LIN {X 0,Y 211.438,Z 626.963,A -85,B 0,C 180,E1 -20790,E2 -20790} C_VEL
LIN {X 0,Y 211.437,Z 626.323,A -85,B 0,C 180,E1 -20793.812,E2 -20793.812} C_VEL
LIN {X 0,Y 211.828,Z 624.336,A -85,B 0,C 180,E1 -20797.626,E2 -20797.626} C_VEL
LIN {X 0,Y 212.751,Z 620.963,A -85,B 0,C 180,E1 -20801.432,E2 -20801.432} C_VEL
LIN {X 0,Y 214.27,Z 616.102,A -85,B 0,C 180,E1 -20805.212,E2 -20805.212} C_VEL
LIN {X 0,Y 216.148,Z 611.384,A -85,B 0,C 180,E1 -20807.992,E2 -20807.992} C_VEL
LIN {X 0,Y 218.416,Z 604.89,A -85,B 0,C 180,E1 -20811.07,E2 -20811.07} C_VEL
LIN {X 0,Y 221.135,Z 597.399,A -85,B 0,C 180,E1 -20813.905,E2 -20813.905} C_VEL
LIN {X 0,Y 224.235,Z 588.787,A -85,B 0,C 180,E1 -20816.527,E2 -20816.527} C_VEL
LIN {X 0,Y 227.75,Z 578.349,A -85,B 0,C 180,E1 -20819.079,E2 -20819.079} C_VEL
LIN {X 0,Y 231.118,Z 567.814,A -85,B 0,C 180,E1 -20821.128,E2 -20821.128} C_VEL
LIN {X 0,Y 234.172,Z 556.322,A -85,B 0,C 180,E1 -20822.954,E2 -20822.954} C_VEL
LIN {X 0,Y 234.795,Z 553.459,A -85,B 0,C 180,E1 -20823.368,E2 -20823.368} C_VEL
LIN {X 0,Y 234.361,Z 541.271,A -85,B 0,C 180,E1 -20825.351,E2 -20825.351} C_VEL
LIN {X 0,Y 232.923,Z 528.444,A -85,B 0,C 180,E1 -20827.232,E2 -20827.232} C_VEL
LIN {X 0,Y 230.563,Z 516.355,A -85,B 0,C 180,E1 -20828.886,E2 -20828.886} C_VEL
LIN {X 0,Y 227.516,Z 504.968,A -85,B 0,C 180,E1 -20830.356,E2 -20830.356} C_VEL
LIN {X 0,Y 222.858,Z 491.263,A -85,B 0,C 180,E1 -20832.099,E2 -20832.099} C_VEL
LIN {X 0,Y 223.254,Z 487.862,A -85,B 0,C 180,E1 -20833.833,E2 -20833.833} C_VEL
LIN {X 0,Y 222.449,Z 481.719,A -85,B 0,C 180,E1 -20837.469,E2 -20837.469} C_VEL
LIN {X 0,Y 221.31,Z 475.041,A -85,B 0,C 180,E1 -20841.74,E2 -20841.74} C_VEL
LIN {X 0,Y 220.41,Z 470.31,A -85,B 0,C 180,E1 -20844.974,E2 -20844.974} C_VEL
LIN {X 0,Y 219.512,Z 466.3,A -85,B 0,C 180,E1 -20847.926,E2 -20847.926} C_VEL
LIN {X 0,Y 222.724,Z 476.254,A -85,B 0,C 180,E1 -20849.677,E2 -20849.677} C_VEL
LIN {X 0,Y 225.072,Z 485.139,A -85,B 0,C 180,E1 -20851.347,E2 -20851.347} C_VEL
LIN {X 0,Y 222.609,Z 498.639,A -85,B 0,C 180,E1 -20853.769,E2 -20853.769} C_VEL
LIN {X 0,Y 220.199,Z 511.207,A -85,B 0,C 180,E1 -20856.487,E2 -20856.487} C_VEL
LIN {X 0,Y 217.759,Z 523.017,A -85,B 0,C 180,E1 -20859.555,E2 -20859.555} C_VEL
LIN {X 0,Y 216.268,Z 532.38,A -85,B 0,C 180,E1 -20862.506,E2 -20862.506} C_VEL
LIN {X 0,Y 214.739,Z 541.158,A -85,B 0,C 180,E1 -20865.791,E2 -20865.791} C_VEL
LIN {X 0,Y 213.615,Z 549.495,A -85,B 0,C 180,E1 -20869.575,E2 -20869.575} C_VEL
LIN {X 0,Y 213.008,Z 556.211,A -85,B 0,C 180,E1 -20873.369,E2 -20873.369} C_VEL
LIN {X 0,Y 212.724,Z 561.483,A -85,B 0,C 180,E1 -20877.159,E2 -20877.159} C_VEL
LIN {X 0,Y 212.687,Z 564.579,A -85,B 0,C 180,E1 -20880,E2 -20880} C_VEL
LIN {X 0,Y 213.289,Z 567.702,A -85,B 0,C 180,E1 -20883.778,E2 -20883.778} C_VEL
LIN {X 0,Y 214.604,Z 569.684,A -85,B 0,C 180,E1 -20887.527,E2 -20887.527} C_VEL
LIN {X 0,Y 216.505,Z 570.581,A -85,B 0,C 180,E1 -20891.231,E2 -20891.231} C_VEL
LIN {X 0,Y 218.953,Z 570.405,A -85,B 0,C 180,E1 -20894.879,E2 -20894.879} C_VEL
LIN {X 0,Y 222.069,Z 569.211,A -85,B 0,C 180,E1 -20898.45,E2 -20898.45} C_VEL
LIN {X 0,Y 226.094,Z 566.97,A -85,B 0,C 180,E1 -20901.901,E2 -20901.901} C_VEL
LIN {X 0,Y 230.851,Z 563.736,A -85,B 0,C 180,E1 -20905.227,E2 -20905.227} C_VEL
LIN {X 0,Y 236.622,Z 559.339,A -85,B 0,C 180,E1 -20908.374,E2 -20908.374} C_VEL
LIN {X 0,Y 244.707,Z 552.327,A -85,B 0,C 180,E1 -20912.095,E2 -20912.095} C_VEL
LIN {X 0,Y 251.951,Z 545.424,A -85,B 0,C 180,E1 -20914.878,E2 -20914.878} C_VEL
LIN {X 0,Y 261.05,Z 536.046,A -85,B 0,C 180,E1 -20917.769,E2 -20917.769} C_VEL
LIN {X 0,Y 264.355,Z 532.395,A -85,B 0,C 180,E1 -20918.706,E2 -20918.706} C_VEL
LIN {X 0,Y 264.555,Z 531.824,A -85,B 0,C 180,E1 -20919.611,E2 -20919.611} C_VEL
LIN {X 0,Y 263.168,Z 532.972,A -85,B 0,C 180,E1 -20921.427,E2 -20921.427} C_VEL
LIN {X 0,Y 262.284,Z 533.945,A -85,B 0,C 180,E1 -20922.232,E2 -20922.232} C_VEL
LIN {X 0,Y 260.132,Z 536.442,A -85,B 0,C 180,E1 -20923.31,E2 -20923.31} C_VEL
LIN {X 0,Y 257.399,Z 539.583,A -85,B 0,C 180,E1 -20924.267,E2 -20924.267} C_VEL
LIN {X 0,Y 251.606,Z 546.399,A -85,B 0,C 180,E1 -20926.185,E2 -20926.185} C_VEL
LIN {X 0,Y 250.054,Z 548.43,A -85,B 0,C 180,E1 -20926.914,E2 -20926.914} C_VEL
LIN {X 0,Y 246.157,Z 553.947,A -85,B 0,C 180,E1 -20928.954,E2 -20928.954} C_VEL
LIN {X 0,Y 241.773,Z 559.648,A -85,B 0,C 180,E1 -20930.784,E2 -20930.784} C_VEL
LIN {X 0,Y 234.168,Z 569.412,A -85,B 0,C 180,E1 -20934.129,E2 -20934.129} C_VEL
LIN {X 0,Y 230.572,Z 573.702,A -85,B 0,C 180,E1 -20935.675,E2 -20935.675} C_VEL
LIN {X 0,Y 223.777,Z 581.401,A -85,B 0,C 180,E1 -20938.788,E2 -20938.788} C_VEL
LIN {X 0,Y 219.264,Z 586.498,A -85,B 0,C 180,E1 -20941.263,E2 -20941.263} C_VEL
LIN {X 0,Y 215.793,Z 596.139,A -85,B 0,C 180,E1 -20943.917,E2 -20943.917} C_VEL
LIN {X 0,Y 212.769,Z 604.113,A -85,B 0,C 180,E1 -20946.648,E2 -20946.648} C_VEL
LIN {X 0,Y 210.282,Z 610.951,A -85,B 0,C 180,E1 -20949.563,E2 -20949.563} C_VEL
LIN {X 0,Y 207.74,Z 617.843,A -85,B 0,C 180,E1 -20953.288,E2 -20953.288} C_VEL
LIN {X 0,Y 206.203,Z 621.981,A -85,B 0,C 180,E1 -20956.197,E2 -20956.197} C_VEL
LIN {X 0,Y 205.043,Z 626.152,A -85,B 0,C 180,E1 -20960.132,E2 -20960.132} C_VEL
LIN {X 0,Y 204.418,Z 628.876,A -85,B 0,C 180,E1 -20964.08,E2 -20964.08} C_VEL
LIN {X 0,Y 204.354,Z 630.227,A -85,B 0,C 180,E1 -20968.029,E2 -20968.029} C_VEL
LIN {X 0,Y 204.409,Z 630.393,A -85,B 0,C 180,E1 -20970,E2 -20970} C_VEL
LIN {X 0,Y 204.342,Z 629.707,A -85,B 0,C 180,E1 -20973.944,E2 -20973.944} C_VEL
LIN {X 0,Y 204.656,Z 627.663,A -85,B 0,C 180,E1 -20977.895,E2 -20977.895} C_VEL
LIN {X 0,Y 205.528,Z 624.213,A -85,B 0,C 180,E1 -20981.839,E2 -20981.839} C_VEL
LIN {X 0,Y 207.176,Z 619.255,A -85,B 0,C 180,E1 -20985.747,E2 -20985.747} C_VEL
LIN {X 0,Y 209.597,Z 612.64,A -85,B 0,C 180,E1 -20989.591,E2 -20989.591} C_VEL
LIN {X 0,Y 212.31,Z 605.237,A -85,B 0,C 180,E1 -20992.89,E2 -20992.89} C_VEL
LIN {X 0,Y 215.211,Z 597.487,A -85,B 0,C 180,E1 -20995.639,E2 -20995.639} C_VEL
LIN {X 0,Y 218.575,Z 588.126,A -85,B 0,C 180,E1 -20998.312,E2 -20998.312} C_VEL
LIN {X 0,Y 222.173,Z 577.744,A -85,B 0,C 180,E1 -21000.669,E2 -21000.669} C_VEL
LIN {X 0,Y 225.594,Z 566.096,A -85,B 0,C 180,E1 -21002.807,E2 -21002.807} C_VEL
LIN {X 0,Y 226.328,Z 562.297,A -85,B 0,C 180,E1 -21003.462,E2 -21003.462} C_VEL
LIN {X 0,Y 226.815,Z 549.482,A -85,B 0,C 180,E1 -21005.641,E2 -21005.641} C_VEL
LIN {X 0,Y 226.84,Z 537.154,A -85,B 0,C 180,E1 -21007.405,E2 -21007.405} C_VEL
LIN {X 0,Y 226.401,Z 530.775,A -85,B 0,C 180,E1 -21008.26,E2 -21008.26} C_VEL
LIN {X 0,Y 224.229,Z 518.623,A -85,B 0,C 180,E1 -21009.922,E2 -21009.922} C_VEL
LIN {X 0,Y 220.801,Z 506.177,A -85,B 0,C 180,E1 -21011.592,E2 -21011.592} C_VEL
LIN {X 0,Y 215.62,Z 492.28,A -85,B 0,C 180,E1 -21013.512,E2 -21013.512} C_VEL
LIN {X 0,Y 214.945,Z 490.339,A -85,B 0,C 180,E1 -21013.832,E2 -21013.832} C_VEL
LIN {X 0,Y 214.514,Z 480.599,A -85,B 0,C 180,E1 -21017.351,E2 -21017.351} C_VEL
LIN {X 0,Y 214.229,Z 476.35,A -85,B 0,C 180,E1 -21018.995,E2 -21018.995} C_VEL
LIN {X 0,Y 213.411,Z 471.066,A -85,B 0,C 180,E1 -21021.266,E2 -21021.266} C_VEL
LIN {X 0,Y 211.376,Z 462.983,A -85,B 0,C 180,E1 -21025.582,E2 -21025.582} C_VEL
LIN {X 0,Y 209.379,Z 455.238,A -85,B 0,C 180,E1 -21030.776,E2 -21030.776} C_VEL
LIN {X 0,Y 208.75,Z 452.356,A -85,B 0,C 180,E1 -21032.967,E2 -21032.967} C_VEL
LIN {X 0,Y 206.768,Z 448.394,A -85,B 0,C 180,E1 -21037.888,E2 -21037.888} C_VEL
LIN {X 0,Y 206.875,Z 448.342,A -85,B 0,C 180,E1 -21042.197,E2 -21042.197} C_VEL
LIN {X 0,Y 206.896,Z 448.315,A -85,B 0,C 180,E1 -21046.245,E2 -21046.245} C_VEL
LIN {X 0,Y 207.101,Z 448.287,A -85,B 0,C 180,E1 -21050.231,E2 -21050.231} C_VEL
LIN {X 0,Y 207.06,Z 448.319,A -85,B 0,C 180,E1 -21054.156,E2 -21054.156} C_VEL
LIN {X 0,Y 207.383,Z 448.253,A -85,B 0,C 180,E1 -21058.058,E2 -21058.058} C_VEL
LIN {X 0,Y 207.521,Z 448.262,A -85,B 0,C 180,E1 -21060,E2 -21060} C_VEL
LIN {X 0,Y 207.384,Z 448.254,A -85,B 0,C 180,E1 -21061.942,E2 -21061.942} C_VEL
LIN {X 0,Y 207.17,Z 448.281,A -85,B 0,C 180,E1 -21067.799,E2 -21067.799} C_VEL
LIN {X 0,Y 207.099,Z 448.398,A -85,B 0,C 180,E1 -21070.221,E2 -21070.221} C_VEL
LIN {X 0,Y 208.263,Z 452.322,A -85,B 0,C 180,E1 -21075.662,E2 -21075.662} C_VEL
LIN {X 0,Y 209.467,Z 456.172,A -85,B 0,C 180,E1 -21080.04,E2 -21080.04} C_VEL
LIN {X 0,Y 211.1,Z 461.213,A -85,B 0,C 180,E1 -21085.111,E2 -21085.111} C_VEL
LIN {X 0,Y 212.2,Z 465.263,A -85,B 0,C 180,E1 -21088.701,E2 -21088.701} C_VEL
LIN {X 0,Y 213.439,Z 470.511,A -85,B 0,C 180,E1 -21092.909,E2 -21092.909} C_VEL
LIN {X 0,Y 214.759,Z 477.132,A -85,B 0,C 180,E1 -21097.715,E2 -21097.715} C_VEL
LIN {X 0,Y 215.772,Z 483.666,A -85,B 0,C 180,E1 -21102.008,E2 -21102.008} C_VEL
LIN {X 0,Y 216.536,Z 489.484,A -85,B 0,C 180,E1 -21105.565,E2 -21105.565} C_VEL
LIN {X 0,Y 216.625,Z 491.594,A -85,B 0,C 180,E1 -21106.615,E2 -21106.615} C_VEL
LIN {X 0,Y 221.782,Z 506.594,A -85,B 0,C 180,E1 -21108.644,E2 -21108.644} C_VEL
LIN {X 0,Y 225.21,Z 519.727,A -85,B 0,C 180,E1 -21110.476,E2 -21110.476} C_VEL
LIN {X 0,Y 227.333,Z 532.987,A -85,B 0,C 180,E1 -21112.391,E2 -21112.391} C_VEL
LIN {X 0,Y 228.381,Z 544.562,A -85,B 0,C 180,E1 -21114.219,E2 -21114.219} C_VEL
LIN {X 0,Y 228.534,Z 554.212,A -85,B 0,C 180,E1 -21115.859,E2 -21115.859} C_VEL
LIN {X 0,Y 225.685,Z 565.569,A -85,B 0,C 180,E1 -21117.654,E2 -21117.654} C_VEL
LIN {X 0,Y 222.371,Z 575.953,A -85,B 0,C 180,E1 -21119.624,E2 -21119.624} C_VEL
LIN {X 0,Y 219.166,Z 585.16,A -85,B 0,C 180,E1 -21121.772,E2 -21121.772} C_VEL
LIN {X 0,Y 215.779,Z 594.41,A -85,B 0,C 180,E1 -21124.434,E2 -21124.434} C_VEL
LIN {X 0,Y 212.744,Z 602.081,A -85,B 0,C 180,E1 -21127.16,E2 -21127.16} C_VEL
LIN {X 0,Y 210.066,Z 609.411,A -85,B 0,C 180,E1 -21130.454,E2 -21130.454} C_VEL
LIN {X 0,Y 208.097,Z 614.497,A -85,B 0,C 180,E1 -21133.317,E2 -21133.317} C_VEL
LIN {X 0,Y 206.152,Z 619.826,A -85,B 0,C 180,E1 -21137.197,E2 -21137.197} C_VEL
LIN {X 0,Y 205.209,Z 622.769,A -85,B 0,C 180,E1 -21140.14,E2 -21140.14} C_VEL
LIN {X 0,Y 204.504,Z 625.484,A -85,B 0,C 180,E1 -21144.082,E2 -21144.082} C_VEL
LIN {X 0,Y 204.306,Z 626.842,A -85,B 0,C 180,E1 -21148.029,E2 -21148.029} C_VEL
LIN {X 0,Y 204.342,Z 627.022,A -85,B 0,C 180,E1 -21150,E2 -21150} C_VEL
LIN {X 0,Y 204.34,Z 626.381,A -85,B 0,C 180,E1 -21153.944,E2 -21153.944} C_VEL
LIN {X 0,Y 204.767,Z 624.394,A -85,B 0,C 180,E1 -21157.891,E2 -21157.891} C_VEL
LIN {X 0,Y 205.778,Z 621.02,A -85,B 0,C 180,E1 -21161.825,E2 -21161.825} C_VEL
LIN {X 0,Y 207.41,Z 616.158,A -85,B 0,C 180,E1 -21165.728,E2 -21165.728} C_VEL
LIN {X 0,Y 209.374,Z 611.44,A -85,B 0,C 180,E1 -21168.595,E2 -21168.595} C_VEL
LIN {X 0,Y 211.569,Z 605.461,A -85,B 0,C 180,E1 -21171.546,E2 -21171.546} C_VEL
LIN {X 0,Y 214.652,Z 597.451,A -85,B 0,C 180,E1 -21174.674,E2 -21174.674} C_VEL
LIN {X 0,Y 217.873,Z 588.837,A -85,B 0,C 180,E1 -21177.366,E2 -21177.366} C_VEL
LIN {X 0,Y 221.568,Z 578.396,A -85,B 0,C 180,E1 -21179.972,E2 -21179.972} C_VEL
LIN {X 0,Y 225.067,Z 567.857,A -85,B 0,C 180,E1 -21182.063,E2 -21182.063} C_VEL
LIN {X 0,Y 228.23,Z 556.361,A -85,B 0,C 180,E1 -21183.927,E2 -21183.927} C_VEL
LIN {X 0,Y 228.579,Z 553.496,A -85,B 0,C 180,E1 -21184.4,E2 -21184.4} C_VEL
LIN {X 0,Y 228.206,Z 541.3,A -85,B 0,C 180,E1 -21186.455,E2 -21186.455} C_VEL
LIN {X 0,Y 226.962,Z 529.515,A -85,B 0,C 180,E1 -21188.266,E2 -21188.266} C_VEL
LIN {X 0,Y 224.537,Z 516.658,A -85,B 0,C 180,E1 -21190.111,E2 -21190.111} C_VEL
LIN {X 0,Y 220.994,Z 503.765,A -85,B 0,C 180,E1 -21191.882,E2 -21191.882} C_VEL
LIN {X 0,Y 216.582,Z 491.242,A -85,B 0,C 180,E1 -21193.619,E2 -21193.619} C_VEL
LIN {X 0,Y 216.312,Z 487.047,A -85,B 0,C 180,E1 -21196.059,E2 -21196.059} C_VEL
LIN {X 0,Y 215.265,Z 480.132,A -85,B 0,C 180,E1 -21200.458,E2 -21200.458} C_VEL
LIN {X 0,Y 214.432,Z 475.169,A -85,B 0,C 180,E1 -21203.846,E2 -21203.846} C_VEL
LIN {X 0,Y 213.284,Z 469.78,A -85,B 0,C 180,E1 -21207.883,E2 -21207.883} C_VEL
LIN {X 0,Y 216.482,Z 480.115,A -85,B 0,C 180,E1 -21209.811,E2 -21209.811} C_VEL
LIN {X 0,Y 217.866,Z 485.033,A -85,B 0,C 180,E1 -21210.778,E2 -21210.778} C_VEL
LIN {X 0,Y 218.03,Z 486.631,A -85,B 0,C 180,E1 -21211.085,E2 -21211.085} C_VEL
LIN {X 0,Y 215.429,Z 500.184,A -85,B 0,C 180,E1 -21213.609,E2 -21213.609} C_VEL
LIN {X 0,Y 213.202,Z 511.621,A -85,B 0,C 180,E1 -21216.183,E2 -21216.183} C_VEL
LIN {X 0,Y 210.832,Z 522.696,A -85,B 0,C 180,E1 -21219.142,E2 -21219.142} C_VEL
LIN {X 0,Y 209.161,Z 532.832,A -85,B 0,C 180,E1 -21222.398,E2 -21222.398} C_VEL
LIN {X 0,Y 207.624,Z 541.695,A -85,B 0,C 180,E1 -21225.794,E2 -21225.794} C_VEL
LIN {X 0,Y 206.589,Z 549.119,A -85,B 0,C 180,E1 -21229.216,E2 -21229.216} C_VEL
LIN {X 0,Y 205.94,Z 556.05,A -85,B 0,C 180,E1 -21233.14,E2 -21233.14} C_VEL
LIN {X 0,Y 205.632,Z 561.568,A -85,B 0,C 180,E1 -21237.061,E2 -21237.061} C_VEL
LIN {X 0,Y 205.594,Z 564.882,A -85,B 0,C 180,E1 -21240,E2 -21240} C_VEL
LIN {X 0,Y 206.245,Z 568.225,A -85,B 0,C 180,E1 -21243.908,E2 -21243.908} C_VEL
LIN {X 0,Y 207.61,Z 570.414,A -85,B 0,C 180,E1 -21247.782,E2 -21247.782} C_VEL
LIN {X 0,Y 209.601,Z 571.515,A -85,B 0,C 180,E1 -21251.606,E2 -21251.606} C_VEL
LIN {X 0,Y 212.196,Z 571.593,A -85,B 0,C 180,E1 -21255.365,E2 -21255.365} C_VEL
LIN {X 0,Y 215.498,Z 570.689,A -85,B 0,C 180,E1 -21259.034,E2 -21259.034} C_VEL
LIN {X 0,Y 219.742,Z 568.777,A -85,B 0,C 180,E1 -21262.569,E2 -21262.569} C_VEL
LIN {X 0,Y 224.734,Z 565.837,A -85,B 0,C 180,E1 -21265.964,E2 -21265.964} C_VEL
LIN {X 0,Y 232.366,Z 560.589,A -85,B 0,C 180,E1 -21269.937,E2 -21269.937} C_VEL
LIN {X 0,Y 239.216,Z 555.235,A -85,B 0,C 180,E1 -21272.923,E2 -21272.923} C_VEL
LIN {X 0,Y 246.751,Z 548.813,A -85,B 0,C 180,E1 -21275.724,E2 -21275.724} C_VEL
LIN {X 0,Y 255.077,Z 541.106,A -85,B 0,C 180,E1 -21278.311,E2 -21278.311} C_VEL
LIN {X 0,Y 259.395,Z 536.877,A -85,B 0,C 180,E1 -21279.505,E2 -21279.505} C_VEL
LIN {X 0,Y 258.265,Z 537.737,A -85,B 0,C 180,E1 -21280.897,E2 -21280.897} C_VEL
LIN {X 0,Y 256.735,Z 539.399,A -85,B 0,C 180,E1 -21282.344,E2 -21282.344} C_VEL
LIN {X 0,Y 254.454,Z 542.279,A -85,B 0,C 180,E1 -21284.1,E2 -21284.1} C_VEL
LIN {X 0,Y 251.189,Z 546.789,A -85,B 0,C 180,E1 -21286.229,E2 -21286.229} C_VEL
LIN {X 0,Y 250.054,Z 548.43,A -85,B 0,C 180,E1 -21286.914,E2 -21286.914} C_VEL
LIN {X 0,Y 247.516,Z 551.631,A -85,B 0,C 180,E1 -21287.904,E2 -21287.904} C_VEL
LIN {X 0,Y 244.193,Z 555.188,A -85,B 0,C 180,E1 -21288.711,E2 -21288.711} C_VEL
LIN {X 0,Y 236.72,Z 562.348,A -85,B 0,C 180,E1 -21290.185,E2 -21290.185} C_VEL
LIN {X 0,Y 233.317,Z 565.671,A -85,B 0,C 180,E1 -21291.079,E2 -21291.079} C_VEL
LIN {X 0,Y 232.346,Z 566.703,A -85,B 0,C 180,E1 -21291.427,E2 -21291.427} C_VEL
LIN {X 0,Y 226.804,Z 573.083,A -85,B 0,C 180,E1 -21293.931,E2 -21293.931} C_VEL
LIN {X 0,Y 219.432,Z 580.604,A -85,B 0,C 180,E1 -21297.011,E2 -21297.011} C_VEL
LIN {X 0,Y 212.547,Z 587.788,A -85,B 0,C 180,E1 -21300.674,E2 -21300.674} C_VEL
LIN {X 0,Y 208.862,Z 597.556,A -85,B 0,C 180,E1 -21303.522,E2 -21303.522} C_VEL
LIN {X 0,Y 205.767,Z 605.284,A -85,B 0,C 180,E1 -21306.339,E2 -21306.339} C_VEL
LIN {X 0,Y 202.966,Z 612.661,A -85,B 0,C 180,E1 -21309.741,E2 -21309.741} C_VEL
LIN {X 0,Y 200.323,Z 619.258,A -85,B 0,C 180,E1 -21313.7,E2 -21313.7} C_VEL
LIN {X 0,Y 198.561,Z 624.197,A -85,B 0,C 180,E1 -21317.739,E2 -21317.739} C_VEL
LIN {X 0,Y 197.603,Z 627.631,A -85,B 0,C 180,E1 -21321.821,E2 -21321.821} C_VEL
LIN {X 0,Y 197.247,Z 629.72,A -85,B 0,C 180,E1 -21326.074,E2 -21326.074} C_VEL
LIN {X 0,Y 197.313,Z 630.335,A -85,B 0,C 180,E1 -21330,E2 -21330} C_VEL
LIN {X 0,Y 197.255,Z 629.648,A -85,B 0,C 180,E1 -21334.086,E2 -21334.086} C_VEL
LIN {X 0,Y 197.598,Z 627.604,A -85,B 0,C 180,E1 -21338.179,E2 -21338.179} C_VEL
LIN {X 0,Y 198.548,Z 624.154,A -85,B 0,C 180,E1 -21342.262,E2 -21342.262} C_VEL
LIN {X 0,Y 200.303,Z 619.196,A -85,B 0,C 180,E1 -21346.302,E2 -21346.302} C_VEL
LIN {X 0,Y 202.867,Z 612.582,A -85,B 0,C 180,E1 -21350.269,E2 -21350.269} C_VEL
LIN {X 0,Y 205.735,Z 605.18,A -85,B 0,C 180,E1 -21353.665,E2 -21353.665} C_VEL
LIN {X 0,Y 208.808,Z 597.431,A -85,B 0,C 180,E1 -21356.485,E2 -21356.485} C_VEL
LIN {X 0,Y 212.316,Z 588.071,A -85,B 0,C 180,E1 -21359.226,E2 -21359.226} C_VEL
LIN {X 0,Y 216.092,Z 577.691,A -85,B 0,C 180,E1 -21361.63,E2 -21361.63} C_VEL
LIN {X 0,Y 219.527,Z 566.482,A -85,B 0,C 180,E1 -21363.741,E2 -21363.741} C_VEL
LIN {X 0,Y 220.172,Z 562.326,A -85,B 0,C 180,E1 -21364.512,E2 -21364.512} C_VEL
LIN {X 0,Y 220.816,Z 549.437,A -85,B 0,C 180,E1 -21366.765,E2 -21366.765} C_VEL
LIN {X 0,Y 220.938,Z 535.461,A -85,B 0,C 180,E1 -21368.801,E2 -21368.801} C_VEL
LIN {X 0,Y 219.026,Z 522.428,A -85,B 0,C 180,E1 -21370.706,E2 -21370.706} C_VEL
LIN {X 0,Y 215.908,Z 509.995,A -85,B 0,C 180,E1 -21372.494,E2 -21372.494} C_VEL
LIN {X 0,Y 211.415,Z 497.153,A -85,B 0,C 180,E1 -21374.379,E2 -21374.379} C_VEL
LIN {X 0,Y 208.837,Z 490.439,A -85,B 0,C 180,E1 -21375.455,E2 -21375.455} C_VEL
LIN {X 0,Y 208.607,Z 482.072,A -85,B 0,C 180,E1 -21378.666,E2 -21378.666} C_VEL
LIN {X 0,Y 207.966,Z 475.685,A -85,B 0,C 180,E1 -21381.43,E2 -21381.43} C_VEL
LIN {X 0,Y 205.88,Z 466.99,A -85,B 0,C 180,E1 -21386.235,E2 -21386.235} C_VEL
LIN {X 0,Y 204.123,Z 459.761,A -85,B 0,C 180,E1 -21391.182,E2 -21391.182} C_VEL
LIN {X 0,Y 203.521,Z 457.099,A -85,B 0,C 180,E1 -21393.326,E2 -21393.326} C_VEL
LIN {X 0,Y 201.76,Z 453.739,A -85,B 0,C 180,E1 -21397.47,E2 -21397.47} C_VEL
LIN {X 0,Y 200.013,Z 450.197,A -85,B 0,C 180,E1 -21403.674,E2 -21403.674} C_VEL
LIN {X 0,Y 199.876,Z 449.189,A -85,B 0,C 180,E1 -21406.27,E2 -21406.27} C_VEL
LIN {X 0,Y 200.024,Z 449.17,A -85,B 0,C 180,E1 -21409.882,E2 -21409.882} C_VEL
LIN {X 0,Y 200.022,Z 449.195,A -85,B 0,C 180,E1 -21413.949,E2 -21413.949} C_VEL
LIN {X 0,Y 200.322,Z 449.131,A -85,B 0,C 180,E1 -21417.99,E2 -21417.99} C_VEL
LIN {X 0,Y 200.485,Z 449.138,A -85,B 0,C 180,E1 -21420,E2 -21420} C_VEL
LIN {X 0,Y 200.18,Z 449.279,A -85,B 0,C 180,E1 -21423.019,E2 -21423.019} C_VEL
LIN {X 0,Y 201.281,Z 452.427,A -85,B 0,C 180,E1 -21430.054,E2 -21430.054} C_VEL
LIN {X 0,Y 202.45,Z 456.655,A -85,B 0,C 180,E1 -21436.124,E2 -21436.124} C_VEL
LIN {X 0,Y 203.541,Z 460.211,A -85,B 0,C 180,E1 -21440.199,E2 -21440.199} C_VEL
LIN {X 0,Y 204.759,Z 464.095,A -85,B 0,C 180,E1 -21444.323,E2 -21444.323} C_VEL
LIN {X 0,Y 206.006,Z 468.65,A -85,B 0,C 180,E1 -21448.53,E2 -21448.53} C_VEL
LIN {X 0,Y 207.159,Z 473.862,A -85,B 0,C 180,E1 -21452.875,E2 -21452.875} C_VEL
LIN {X 0,Y 208.341,Z 479.943,A -85,B 0,C 180,E1 -21457.387,E2 -21457.387} C_VEL
LIN {X 0,Y 209.382,Z 487.02,A -85,B 0,C 180,E1 -21462.168,E2 -21462.168} C_VEL
LIN {X 0,Y 209.967,Z 491.492,A -85,B 0,C 180,E1 -21464.87,E2 -21464.87} C_VEL
LIN {X 0,Y 212.48,Z 496.88,A -85,B 0,C 180,E1 -21465.799,E2 -21465.799} C_VEL
LIN {X 0,Y 216.985,Z 510.929,A -85,B 0,C 180,E1 -21467.837,E2 -21467.837} C_VEL
LIN {X 0,Y 219.906,Z 523.685,A -85,B 0,C 180,E1 -21469.732,E2 -21469.732} C_VEL
LIN {X 0,Y 221.641,Z 536.427,A -85,B 0,C 180,E1 -21471.702,E2 -21471.702} C_VEL
LIN {X 0,Y 222.411,Z 548.224,A -85,B 0,C 180,E1 -21473.695,E2 -21473.695} C_VEL
LIN {X 0,Y 222.341,Z 555.692,A -85,B 0,C 180,E1 -21475.051,E2 -21475.051} C_VEL
LIN {X 0,Y 219.19,Z 567.292,A -85,B 0,C 180,E1 -21476.97,E2 -21476.97} C_VEL
LIN {X 0,Y 215.544,Z 577.935,A -85,B 0,C 180,E1 -21479.1,E2 -21479.1} C_VEL
LIN {X 0,Y 211.663,Z 588.462,A -85,B 0,C 180,E1 -21481.761,E2 -21481.761} C_VEL
LIN {X 0,Y 208.241,Z 597.148,A -85,B 0,C 180,E1 -21484.513,E2 -21484.513} C_VEL
LIN {X 0,Y 204.814,Z 605.468,A -85,B 0,C 180,E1 -21487.824,E2 -21487.824} C_VEL
LIN {X 0,Y 202.685,Z 611.255,A -85,B 0,C 180,E1 -21490.767,E2 -21490.767} C_VEL
LIN {X 0,Y 200.088,Z 617.43,A -85,B 0,C 180,E1 -21494.726,E2 -21494.726} C_VEL
LIN {X 0,Y 198.823,Z 620.939,A -85,B 0,C 180,E1 -21497.755,E2 -21497.755} C_VEL
LIN {X 0,Y 197.719,Z 624.359,A -85,B 0,C 180,E1 -21501.826,E2 -21501.826} C_VEL
LIN {X 0,Y 197.243,Z 626.457,A -85,B 0,C 180,E1 -21506.096,E2 -21506.096} C_VEL
LIN {X 0,Y 197.249,Z 627.08,A -85,B 0,C 180,E1 -21510,E2 -21510} C_VEL
LIN {X 0,Y 197.25,Z 626.44,A -85,B 0,C 180,E1 -21514.086,E2 -21514.086} C_VEL
LIN {X 0,Y 197.718,Z 624.452,A -85,B 0,C 180,E1 -21518.174,E2 -21518.174} C_VEL
LIN {X 0,Y 198.802,Z 621.077,A -85,B 0,C 180,E1 -21522.246,E2 -21522.246} C_VEL
LIN {X 0,Y 200.574,Z 616.214,A -85,B 0,C 180,E1 -21526.279,E2 -21526.279} C_VEL
LIN {X 0,Y 202.626,Z 611.495,A -85,B 0,C 180,E1 -21529.239,E2 -21529.239} C_VEL
LIN {X 0,Y 205.291,Z 604.658,A -85,B 0,C 180,E1 -21532.652,E2 -21532.652} C_VEL
LIN {X 0,Y 208.737,Z 596.167,A -85,B 0,C 180,E1 -21535.957,E2 -21535.957} C_VEL
LIN {X 0,Y 212.185,Z 587.283,A -85,B 0,C 180,E1 -21538.703,E2 -21538.703} C_VEL
LIN {X 0,Y 216.16,Z 576.522,A -85,B 0,C 180,E1 -21541.346,E2 -21541.346} C_VEL
LIN {X 0,Y 219.815,Z 565.492,A -85,B 0,C 180,E1 -21543.493,E2 -21543.493} C_VEL
LIN {X 0,Y 222.348,Z 556.398,A -85,B 0,C 180,E1 -21544.953,E2 -21544.953} C_VEL
LIN {X 0,Y 222.362,Z 545.505,A -85,B 0,C 180,E1 -21546.907,E2 -21546.907} C_VEL
LIN {X 0,Y 221.366,Z 533.194,A -85,B 0,C 180,E1 -21548.938,E2 -21548.938} C_VEL
LIN {X 0,Y 219.51,Z 521.652,A -85,B 0,C 180,E1 -21550.721,E2 -21550.721} C_VEL
LIN {X 0,Y 216.944,Z 510.654,A -85,B 0,C 180,E1 -21552.352,E2 -21552.352} C_VEL
LIN {X 0,Y 212.775,Z 497.682,A -85,B 0,C 180,E1 -21554.248,E2 -21554.248} C_VEL
LIN {X 0,Y 211.482,Z 494.592,A -85,B 0,C 180,E1 -21554.739,E2 -21554.739} C_VEL
LIN {X 0,Y 209.967,Z 491.274,A -85,B 0,C 180,E1 -21555.339,E2 -21555.339} C_VEL
LIN {X 0,Y 209.208,Z 485.376,A -85,B 0,C 180,E1 -21559.075,E2 -21559.075} C_VEL
LIN {X 0,Y 208.025,Z 478.03,A -85,B 0,C 180,E1 -21564.177,E2 -21564.177} C_VEL
LIN {X 0,Y 207.124,Z 473.331,A -85,B 0,C 180,E1 -21567.916,E2 -21567.916} C_VEL
LIN {X 0,Y 210.551,Z 485.035,A -85,B 0,C 180,E1 -21570.211,E2 -21570.211} C_VEL
LIN {X 0,Y 210.99,Z 487.848,A -85,B 0,C 180,E1 -21570.781,E2 -21570.781} C_VEL
LIN {X 0,Y 208.496,Z 500.373,A -85,B 0,C 180,E1 -21573.202,E2 -21573.202} C_VEL
LIN {X 0,Y 206.214,Z 511.892,A -85,B 0,C 180,E1 -21575.859,E2 -21575.859} C_VEL
LIN {X 0,Y 203.923,Z 522.329,A -85,B 0,C 180,E1 -21578.697,E2 -21578.697} C_VEL
LIN {X 0,Y 202.335,Z 531.874,A -85,B 0,C 180,E1 -21581.783,E2 -21581.783} C_VEL
LIN {X 0,Y 200.677,Z 540.99,A -85,B 0,C 180,E1 -21585.291,E2 -21585.291} C_VEL
LIN {X 0,Y 199.566,Z 548.646,A -85,B 0,C 180,E1 -21588.832,E2 -21588.832} C_VEL
LIN {X 0,Y 198.856,Z 555.851,A -85,B 0,C 180,E1 -21592.894,E2 -21592.894} C_VEL
LIN {X 0,Y 198.614,Z 560.314,A -85,B 0,C 180,E1 -21595.942,E2 -21595.942} C_VEL
LIN {X 0,Y 198.497,Z 565.064,A -85,B 0,C 180,E1 -21600,E2 -21600} C_VEL
LIN {X 0,Y 199.186,Z 568.635,A -85,B 0,C 180,E1 -21604.046,E2 -21604.046} C_VEL
LIN {X 0,Y 200.622,Z 571.058,A -85,B 0,C 180,E1 -21608.055,E2 -21608.055} C_VEL
LIN {X 0,Y 202.707,Z 572.433,A -85,B 0,C 180,E1 -21612.006,E2 -21612.006} C_VEL
LIN {X 0,Y 205.457,Z 572.798,A -85,B 0,C 180,E1 -21615.882,E2 -21615.882} C_VEL
LIN {X 0,Y 208.958,Z 572.146,A -85,B 0,C 180,E1 -21619.654,E2 -21619.654} C_VEL
LIN {X 0,Y 213.402,Z 570.472,A -85,B 0,C 180,E1 -21623.278,E2 -21623.278} C_VEL
LIN {X 0,Y 218.652,Z 567.863,A -85,B 0,C 180,E1 -21626.743,E2 -21626.743} C_VEL
LIN {X 0,Y 226.632,Z 563.104,A -85,B 0,C 180,E1 -21630.775,E2 -21630.775} C_VEL
LIN {X 0,Y 235.657,Z 556.786,A -85,B 0,C 180,E1 -21634.516,E2 -21634.516} C_VEL
LIN {X 0,Y 243.699,Z 550.537,A -85,B 0,C 180,E1 -21637.273,E2 -21637.273} C_VEL
LIN {X 0,Y 252.479,Z 543.078,A -85,B 0,C 180,E1 -21639.809,E2 -21639.809} C_VEL
LIN {X 0,Y 253.38,Z 542.216,A -85,B 0,C 180,E1 -21640.327,E2 -21640.327} C_VEL
LIN {X 0,Y 251.195,Z 544.393,A -85,B 0,C 180,E1 -21642.181,E2 -21642.181} C_VEL
LIN {X 0,Y 248.724,Z 547.247,A -85,B 0,C 180,E1 -21643.901,E2 -21643.901} C_VEL
LIN {X 0,Y 244.441,Z 552.537,A -85,B 0,C 180,E1 -21646.367,E2 -21646.367} C_VEL
LIN {X 0,Y 240.375,Z 557.562,A -85,B 0,C 180,E1 -21648.306,E2 -21648.306} C_VEL
LIN {X 0,Y 232.346,Z 566.703,A -85,B 0,C 180,E1 -21651.427,E2 -21651.427} C_VEL
LIN {X 0,Y 229.141,Z 569.833,A -85,B 0,C 180,E1 -21652.404,E2 -21652.404} C_VEL
LIN {X 0,Y 222.536,Z 575.034,A -85,B 0,C 180,E1 -21653.774,E2 -21653.774} C_VEL
LIN {X 0,Y 215.912,Z 579.785,A -85,B 0,C 180,E1 -21655.248,E2 -21655.248} C_VEL
LIN {X 0,Y 212.741,Z 582.343,A -85,B 0,C 180,E1 -21656.383,E2 -21656.383} C_VEL
LIN {X 0,Y 206.018,Z 588.612,A -85,B 0,C 180,E1 -21659.931,E2 -21659.931} C_VEL
LIN {X 0,Y 202.49,Z 597.504,A -85,B 0,C 180,E1 -21662.621,E2 -21662.621} C_VEL
LIN {X 0,Y 199.232,Z 605.23,A -85,B 0,C 180,E1 -21665.513,E2 -21665.513} C_VEL
LIN {X 0,Y 196.27,Z 612.606,A -85,B 0,C 180,E1 -21669.018,E2 -21669.018} C_VEL
LIN {X 0,Y 193.479,Z 619.202,A -85,B 0,C 180,E1 -21673.106,E2 -21673.106} C_VEL
LIN {X 0,Y 191.596,Z 624.139,A -85,B 0,C 180,E1 -21677.286,E2 -21677.286} C_VEL
LIN {X 0,Y 190.548,Z 627.573,A -85,B 0,C 180,E1 -21681.516,E2 -21681.516} C_VEL
LIN {X 0,Y 190.165,Z 629.605,A -85,B 0,C 180,E1 -21685.761,E2 -21685.761} C_VEL
LIN {X 0,Y 190.169,Z 630.11,A -85,B 0,C 180,E1 -21687.882,E2 -21687.882} C_VEL
LIN {X 0,Y 190.219,Z 630.276,A -85,B 0,C 180,E1 -21690,E2 -21690} C_VEL
LIN {X 0,Y 190.165,Z 629.589,A -85,B 0,C 180,E1 -21694.239,E2 -21694.239} C_VEL
LIN {X 0,Y 190.541,Z 627.545,A -85,B 0,C 180,E1 -21698.484,E2 -21698.484} C_VEL
LIN {X 0,Y 191.584,Z 624.095,A -85,B 0,C 180,E1 -21702.715,E2 -21702.715} C_VEL
LIN {X 0,Y 193.459,Z 619.137,A -85,B 0,C 180,E1 -21706.895,E2 -21706.895} C_VEL
LIN {X 0,Y 196.162,Z 612.524,A -85,B 0,C 180,E1 -21710.994,E2 -21710.994} C_VEL
LIN {X 0,Y 199.215,Z 605.122,A -85,B 0,C 180,E1 -21714.489,E2 -21714.489} C_VEL
LIN {X 0,Y 202.428,Z 597.374,A -85,B 0,C 180,E1 -21717.388,E2 -21717.388} C_VEL
LIN {X 0,Y 206.133,Z 588.017,A -85,B 0,C 180,E1 -21720.192,E2 -21720.192} C_VEL
LIN {X 0,Y 210.405,Z 576.662,A -85,B 0,C 180,E1 -21722.851,E2 -21722.851} C_VEL
LIN {X 0,Y 213.644,Z 566.303,A -85,B 0,C 180,E1 -21724.83,E2 -21724.83} C_VEL
LIN {X 0,Y 214.683,Z 553.971,A -85,B 0,C 180,E1 -21727.171,E2 -21727.171} C_VEL
LIN {X 0,Y 215.203,Z 540.437,A -85,B 0,C 180,E1 -21729.332,E2 -21729.332} C_VEL
LIN {X 0,Y 214.726,Z 532.67,A -85,B 0,C 180,E1 -21730.523,E2 -21730.523} C_VEL
LIN {X 0,Y 212.642,Z 520.579,A -85,B 0,C 180,E1 -21732.398,E2 -21732.398} C_VEL
LIN {X 0,Y 209.758,Z 509.54,A -85,B 0,C 180,E1 -21734.087,E2 -21734.087} C_VEL
LIN {X 0,Y 205.509,Z 497.517,A -85,B 0,C 180,E1 -21735.998,E2 -21735.998} C_VEL
LIN {X 0,Y 202.82,Z 490.427,A -85,B 0,C 180,E1 -21737.225,E2 -21737.225} C_VEL
LIN {X 0,Y 202.644,Z 483.258,A -85,B 0,C 180,E1 -21740.204,E2 -21740.204} C_VEL
LIN {X 0,Y 202.281,Z 479.573,A -85,B 0,C 180,E1 -21741.925,E2 -21741.925} C_VEL
LIN {X 0,Y 200.648,Z 472.384,A -85,B 0,C 180,E1 -21745.915,E2 -21745.915} C_VEL
LIN {X 0,Y 198.812,Z 464.347,A -85,B 0,C 180,E1 -21751.497,E2 -21751.497} C_VEL
LIN {X 0,Y 198.52,Z 462.907,A -85,B 0,C 180,E1 -21752.598,E2 -21752.598} C_VEL
LIN {X 0,Y 196.801,Z 459.216,A -85,B 0,C 180,E1 -21756.87,E2 -21756.87} C_VEL
LIN {X 0,Y 195.336,Z 456.405,A -85,B 0,C 180,E1 -21761.107,E2 -21761.107} C_VEL
LIN {X 0,Y 194.664,Z 454.253,A -85,B 0,C 180,E1 -21765.361,E2 -21765.361} C_VEL
LIN {X 0,Y 194.062,Z 453.08,A -85,B 0,C 180,E1 -21769.568,E2 -21769.568} C_VEL
LIN {X 0,Y 193.814,Z 452.628,A -85,B 0,C 180,E1 -21773.755,E2 -21773.755} C_VEL
LIN {X 0,Y 194.09,Z 452.545,A -85,B 0,C 180,E1 -21777.925,E2 -21777.925} C_VEL
LIN {X 0,Y 194.412,Z 452.776,A -85,B 0,C 180,E1 -21780,E2 -21780} C_VEL
LIN {X 0,Y 194.58,Z 453.331,A -85,B 0,C 180,E1 -21782.07,E2 -21782.07} C_VEL
LIN {X 0,Y 195.272,Z 455.957,A -85,B 0,C 180,E1 -21788.277,E2 -21788.277} C_VEL
LIN {X 0,Y 195.659,Z 456.978,A -85,B 0,C 180,E1 -21790.347,E2 -21790.347} C_VEL
LIN {X 0,Y 196.836,Z 461.258,A -85,B 0,C 180,E1 -21796.597,E2 -21796.597} C_VEL
LIN {X 0,Y 197.774,Z 464.718,A -85,B 0,C 180,E1 -21800.815,E2 -21800.815} C_VEL
LIN {X 0,Y 198.952,Z 468.675,A -85,B 0,C 180,E1 -21805.081,E2 -21805.081} C_VEL
LIN {X 0,Y 199.865,Z 472.226,A -85,B 0,C 180,E1 -21808.467,E2 -21808.467} C_VEL
LIN {X 0,Y 200.975,Z 477.463,A -85,B 0,C 180,E1 -21812.937,E2 -21812.937} C_VEL
LIN {X 0,Y 202.023,Z 483.446,A -85,B 0,C 180,E1 -21817.501,E2 -21817.501} C_VEL
LIN {X 0,Y 202.949,Z 489.99,A -85,B 0,C 180,E1 -21822.036,E2 -21822.036} C_VEL
LIN {X 0,Y 203.128,Z 491.347,A -85,B 0,C 180,E1 -21822.894,E2 -21822.894} C_VEL
LIN {X 0,Y 205.196,Z 495.332,A -85,B 0,C 180,E1 -21823.709,E2 -21823.709} C_VEL
LIN {X 0,Y 207.928,Z 500.978,A -85,B 0,C 180,E1 -21824.807,E2 -21824.807} C_VEL
LIN {X 0,Y 211.735,Z 513.8,A -85,B 0,C 180,E1 -21826.802,E2 -21826.802} C_VEL
LIN {X 0,Y 214.483,Z 527.077,A -85,B 0,C 180,E1 -21828.907,E2 -21828.907} C_VEL
LIN {X 0,Y 215.811,Z 538.488,A -85,B 0,C 180,E1 -21830.782,E2 -21830.782} C_VEL
LIN {X 0,Y 216.37,Z 550.453,A -85,B 0,C 180,E1 -21832.918,E2 -21832.918} C_VEL
LIN {X 0,Y 216.205,Z 557.113,A -85,B 0,C 180,E1 -21834.189,E2 -21834.189} C_VEL
LIN {X 0,Y 212.884,Z 568.497,A -85,B 0,C 180,E1 -21836.145,E2 -21836.145} C_VEL
LIN {X 0,Y 208.743,Z 579.91,A -85,B 0,C 180,E1 -21838.543,E2 -21838.543} C_VEL
LIN {X 0,Y 204.798,Z 590.119,A -85,B 0,C 180,E1 -21841.286,E2 -21841.286} C_VEL
LIN {X 0,Y 201.275,Z 598.537,A -85,B 0,C 180,E1 -21844.121,E2 -21844.121} C_VEL
LIN {X 0,Y 197.804,Z 606.462,A -85,B 0,C 180,E1 -21847.487,E2 -21847.487} C_VEL
LIN {X 0,Y 195.228,Z 613.02,A -85,B 0,C 180,E1 -21851.096,E2 -21851.096} C_VEL
LIN {X 0,Y 192.694,Z 618.735,A -85,B 0,C 180,E1 -21855.208,E2 -21855.208} C_VEL
LIN {X 0,Y 191.204,Z 622.887,A -85,B 0,C 180,E1 -21859.41,E2 -21859.41} C_VEL
LIN {X 0,Y 190.363,Z 625.602,A -85,B 0,C 180,E1 -21863.641,E2 -21863.641} C_VEL
LIN {X 0,Y 190.129,Z 626.959,A -85,B 0,C 180,E1 -21867.882,E2 -21867.882} C_VEL
LIN {X 0,Y 190.158,Z 627.139,A -85,B 0,C 180,E1 -21870,E2 -21870} C_VEL
LIN {X 0,Y 190.166,Z 626.498,A -85,B 0,C 180,E1 -21874.239,E2 -21874.239} C_VEL
LIN {X 0,Y 190.69,Z 624.509,A -85,B 0,C 180,E1 -21878.478,E2 -21878.478} C_VEL
LIN {X 0,Y 191.821,Z 621.135,A -85,B 0,C 180,E1 -21882.699,E2 -21882.699} C_VEL
LIN {X 0,Y 193.763,Z 616.27,A -85,B 0,C 180,E1 -21886.868,E2 -21886.868} C_VEL
LIN {X 0,Y 195.892,Z 611.551,A -85,B 0,C 180,E1 -21889.928,E2 -21889.928} C_VEL
LIN {X 0,Y 198.712,Z 604.712,A -85,B 0,C 180,E1 -21893.446,E2 -21893.446} C_VEL
LIN {X 0,Y 202.361,Z 596.219,A -85,B 0,C 180,E1 -21896.839,E2 -21896.839} C_VEL
LIN {X 0,Y 205.952,Z 587.333,A -85,B 0,C 180,E1 -21899.657,E2 -21899.657} C_VEL
LIN {X 0,Y 210.124,Z 576.568,A -85,B 0,C 180,E1 -21902.354,E2 -21902.354} C_VEL
LIN {X 0,Y 213.674,Z 566.274,A -85,B 0,C 180,E1 -21904.409,E2 -21904.409} C_VEL
LIN {X 0,Y 216.159,Z 557.834,A -85,B 0,C 180,E1 -21905.82,E2 -21905.82} C_VEL
LIN {X 0,Y 216.385,Z 547.573,A -85,B 0,C 180,E1 -21907.757,E2 -21907.757} C_VEL
LIN {X 0,Y 215.688,Z 535.921,A -85,B 0,C 180,E1 -21909.792,E2 -21909.792} C_VEL
LIN {X 0,Y 214.063,Z 524.471,A -85,B 0,C 180,E1 -21911.676,E2 -21911.676} C_VEL
LIN {X 0,Y 211.475,Z 512.41,A -85,B 0,C 180,E1 -21913.558,E2 -21913.558} C_VEL
LIN {X 0,Y 207.564,Z 499.808,A -85,B 0,C 180,E1 -21915.535,E2 -21915.535} C_VEL
LIN {X 0,Y 205.097,Z 495.165,A -85,B 0,C 180,E1 -21916.5,E2 -21916.5} C_VEL
LIN {X 0,Y 203.147,Z 491.299,A -85,B 0,C 180,E1 -21917.291,E2 -21917.291} C_VEL
LIN {X 0,Y 202.33,Z 485.378,A -85,B 0,C 180,E1 -21921.3,E2 -21921.3} C_VEL
LIN {X 0,Y 201.581,Z 480.521,A -85,B 0,C 180,E1 -21924.882,E2 -21924.882} C_VEL
LIN {X 0,Y 200.813,Z 476.76,A -85,B 0,C 180,E1 -21927.942,E2 -21927.942} C_VEL
LIN {X 0,Y 203.822,Z 487.245,A -85,B 0,C 180,E1 -21930.116,E2 -21930.116} C_VEL
LIN {X 0,Y 203.961,Z 488.71,A -85,B 0,C 180,E1 -21930.416,E2 -21930.416} C_VEL
LIN {X 0,Y 201.325,Z 501.663,A -85,B 0,C 180,E1 -21933.011,E2 -21933.011} C_VEL
LIN {X 0,Y 198.807,Z 514.089,A -85,B 0,C 180,E1 -21936.012,E2 -21936.012} C_VEL
LIN {X 0,Y 196.537,Z 524.559,A -85,B 0,C 180,E1 -21939.047,E2 -21939.047} C_VEL
LIN {X 0,Y 194.953,Z 533.597,A -85,B 0,C 180,E1 -21942.156,E2 -21942.156} C_VEL
LIN {X 0,Y 193.35,Z 542.565,A -85,B 0,C 180,E1 -21945.797,E2 -21945.797} C_VEL
LIN {X 0,Y 192.234,Z 551.199,A -85,B 0,C 180,E1 -21950.052,E2 -21950.052} C_VEL
LIN {X 0,Y 191.723,Z 557.185,A -85,B 0,C 180,E1 -21953.686,E2 -21953.686} C_VEL
LIN {X 0,Y 191.422,Z 562.838,A -85,B 0,C 180,E1 -21957.896,E2 -21957.896} C_VEL
LIN {X 0,Y 191.692,Z 567.248,A -85,B 0,C 180,E1 -21962.101,E2 -21962.101} C_VEL
LIN {X 0,Y 192.807,Z 570.485,A -85,B 0,C 180,E1 -21966.278,E2 -21966.278} C_VEL
LIN {X 0,Y 194.661,Z 572.646,A -85,B 0,C 180,E1 -21970.4,E2 -21970.4} C_VEL
LIN {X 0,Y 197.173,Z 573.733,A -85,B 0,C 180,E1 -21974.448,E2 -21974.448} C_VEL
LIN {X 0,Y 200.422,Z 573.835,A -85,B 0,C 180,E1 -21978.397,E2 -21978.397} C_VEL
LIN {X 0,Y 204.598,Z 572.978,A -85,B 0,C 180,E1 -21982.201,E2 -21982.201} C_VEL
LIN {X 0,Y 209.772,Z 571.162,A -85,B 0,C 180,E1 -21985.82,E2 -21985.82} C_VEL
LIN {X 0,Y 215.815,Z 568.364,A -85,B 0,C 180,E1 -21989.24,E2 -21989.24} C_VEL
LIN {X 0,Y 224.545,Z 563.445,A -85,B 0,C 180,E1 -21993.211,E2 -21993.211} C_VEL
LIN {X 0,Y 234.391,Z 556.999,A -85,B 0,C 180,E1 -21996.847,E2 -21996.847} C_VEL
LIN {X 0,Y 243.113,Z 550.658,A -85,B 0,C 180,E1 -21999.493,E2 -21999.493} C_VEL
LIN {X 0,Y 245.405,Z 548.913,A -85,B 0,C 180,E1 -22000.118,E2 -22000.118} C_VEL
LIN {X 0,Y 246.972,Z 547.695,A -85,B 0,C 180,E1 -22000.882,E2 -22000.882} C_VEL
LIN {X 0,Y 244.2,Z 550.44,A -85,B 0,C 180,E1 -22002.801,E2 -22002.801} C_VEL
LIN {X 0,Y 241.163,Z 553.717,A -85,B 0,C 180,E1 -22004.54,E2 -22004.54} C_VEL
LIN {X 0,Y 238.01,Z 557.201,A -85,B 0,C 180,E1 -22006.105,E2 -22006.105} C_VEL
LIN {X 0,Y 233.491,Z 562.003,A -85,B 0,C 180,E1 -22007.955,E2 -22007.955} C_VEL
LIN {X 0,Y 223.778,Z 571.9,A -85,B 0,C 180,E1 -22011.735,E2 -22011.735} C_VEL
LIN {X 0,Y 221.215,Z 574.567,A -85,B 0,C 180,E1 -22012.87,E2 -22012.87} C_VEL
LIN {X 0,Y 212.741,Z 582.343,A -85,B 0,C 180,E1 -22016.383,E2 -22016.383} C_VEL
LIN {X 0,Y 210.396,Z 584.072,A -85,B 0,C 180,E1 -22017.162,E2 -22017.162} C_VEL
LIN {X 0,Y 200.336,Z 589.629,A -85,B 0,C 180,E1 -22019.167,E2 -22019.167} C_VEL
LIN {X 0,Y 198.477,Z 591.934,A -85,B 0,C 180,E1 -22019.889,E2 -22019.889} C_VEL
LIN {X 0,Y 195.008,Z 600.154,A -85,B 0,C 180,E1 -22022.645,E2 -22022.645} C_VEL
LIN {X 0,Y 191.262,Z 608.529,A -85,B 0,C 180,E1 -22026.159,E2 -22026.159} C_VEL
LIN {X 0,Y 188.803,Z 614.354,A -85,B 0,C 180,E1 -22029.291,E2 -22029.291} C_VEL
LIN {X 0,Y 186.664,Z 619.145,A -85,B 0,C 180,E1 -22032.47,E2 -22032.47} C_VEL
LIN {X 0,Y 184.629,Z 624.082,A -85,B 0,C 180,E1 -22036.798,E2 -22036.798} C_VEL
LIN {X 0,Y 183.514,Z 627.515,A -85,B 0,C 180,E1 -22041.188,E2 -22041.188} C_VEL
LIN {X 0,Y 183.078,Z 629.546,A -85,B 0,C 180,E1 -22045.597,E2 -22045.597} C_VEL
LIN {X 0,Y 183.127,Z 630.218,A -85,B 0,C 180,E1 -22050,E2 -22050} C_VEL
LIN {X 0,Y 183.078,Z 629.53,A -85,B 0,C 180,E1 -22054.403,E2 -22054.403} C_VEL
LIN {X 0,Y 183.506,Z 627.486,A -85,B 0,C 180,E1 -22058.812,E2 -22058.812} C_VEL
LIN {X 0,Y 184.618,Z 624.036,A -85,B 0,C 180,E1 -22063.203,E2 -22063.203} C_VEL
LIN {X 0,Y 186.642,Z 619.078,A -85,B 0,C 180,E1 -22067.532,E2 -22067.532} C_VEL
LIN {X 0,Y 189.473,Z 612.465,A -85,B 0,C 180,E1 -22071.773,E2 -22071.773} C_VEL
LIN {X 0,Y 192.737,Z 605.065,A -85,B 0,C 180,E1 -22075.37,E2 -22075.37} C_VEL
LIN {X 0,Y 196.109,Z 597.318,A -85,B 0,C 180,E1 -22078.349,E2 -22078.349} C_VEL
LIN {X 0,Y 200.017,Z 587.962,A -85,B 0,C 180,E1 -22081.216,E2 -22081.216} C_VEL
LIN {X 0,Y 204.401,Z 576.792,A -85,B 0,C 180,E1 -22083.893,E2 -22083.893} C_VEL
LIN {X 0,Y 207.497,Z 567.409,A -85,B 0,C 180,E1 -22085.75,E2 -22085.75} C_VEL
LIN {X 0,Y 208.708,Z 555.534,A -85,B 0,C 180,E1 -22088.11,E2 -22088.11} C_VEL
LIN {X 0,Y 209.406,Z 543.047,A -85,B 0,C 180,E1 -22090.218,E2 -22090.218} C_VEL
LIN {X 0,Y 209.192,Z 536.101,A -85,B 0,C 180,E1 -22091.335,E2 -22091.335} C_VEL
LIN {X 0,Y 207.535,Z 524.365,A -85,B 0,C 180,E1 -22093.273,E2 -22093.273} C_VEL
LIN {X 0,Y 204.997,Z 513.359,A -85,B 0,C 180,E1 -22095.087,E2 -22095.087} C_VEL
LIN {X 0,Y 200.963,Z 501.127,A -85,B 0,C 180,E1 -22097.159,E2 -22097.159} C_VEL
LIN {X 0,Y 196.824,Z 490.476,A -85,B 0,C 180,E1 -22099.144,E2 -22099.144} C_VEL
LIN {X 0,Y 196.691,Z 484.562,A -85,B 0,C 180,E1 -22101.821,E2 -22101.821} C_VEL
LIN {X 0,Y 195.094,Z 476.362,A -85,B 0,C 180,E1 -22106.538,E2 -22106.538} C_VEL
LIN {X 0,Y 193.507,Z 468.921,A -85,B 0,C 180,E1 -22111.826,E2 -22111.826} C_VEL
LIN {X 0,Y 193.25,Z 467.523,A -85,B 0,C 180,E1 -22112.961,E2 -22112.961} C_VEL
LIN {X 0,Y 191.813,Z 464.552,A -85,B 0,C 180,E1 -22116.348,E2 -22116.348} C_VEL
LIN {X 0,Y 190.354,Z 461.617,A -85,B 0,C 180,E1 -22120.593,E2 -22120.593} C_VEL
LIN {X 0,Y 189.506,Z 459.336,A -85,B 0,C 180,E1 -22124.954,E2 -22124.954} C_VEL
LIN {X 0,Y 188.848,Z 457.925,A -85,B 0,C 180,E1 -22129.276,E2 -22129.276} C_VEL
LIN {X 0,Y 188.539,Z 457.376,A -85,B 0,C 180,E1 -22133.579,E2 -22133.579} C_VEL
LIN {X 0,Y 188.725,Z 457.211,A -85,B 0,C 180,E1 -22137.866,E2 -22137.866} C_VEL
LIN {X 0,Y 188.97,Z 457.346,A -85,B 0,C 180,E1 -22140,E2 -22140} C_VEL
LIN {X 0,Y 189.049,Z 457.863,A -85,B 0,C 180,E1 -22142.131,E2 -22142.131} C_VEL
LIN {X 0,Y 189.712,Z 460.433,A -85,B 0,C 180,E1 -22148.522,E2 -22148.522} C_VEL
LIN {X 0,Y 190.017,Z 461.511,A -85,B 0,C 180,E1 -22150.657,E2 -22150.657} C_VEL
LIN {X 0,Y 190.998,Z 465.482,A -85,B 0,C 180,E1 -22156.922,E2 -22156.922} C_VEL
LIN {X 0,Y 191.977,Z 469.228,A -85,B 0,C 180,E1 -22161.475,E2 -22161.475} C_VEL
LIN {X 0,Y 193.098,Z 473.229,A -85,B 0,C 180,E1 -22165.897,E2 -22165.897} C_VEL
LIN {X 0,Y 193.96,Z 477.123,A -85,B 0,C 180,E1 -22169.585,E2 -22169.585} C_VEL
LIN {X 0,Y 194.729,Z 480.803,A -85,B 0,C 180,E1 -22172.777,E2 -22172.777} C_VEL
LIN {X 0,Y 195.493,Z 485.328,A -85,B 0,C 180,E1 -22176.383,E2 -22176.383} C_VEL
LIN {X 0,Y 196.39,Z 491.521,A -85,B 0,C 180,E1 -22180.747,E2 -22180.747} C_VEL
LIN {X 0,Y 198.628,Z 495.606,A -85,B 0,C 180,E1 -22181.708,E2 -22181.708} C_VEL
LIN {X 0,Y 202.481,Z 502.809,A -85,B 0,C 180,E1 -22183.354,E2 -22183.354} C_VEL
LIN {X 0,Y 204.016,Z 507.109,A -85,B 0,C 180,E1 -22184.13,E2 -22184.13} C_VEL
LIN {X 0,Y 207.283,Z 519.938,A -85,B 0,C 180,E1 -22186.271,E2 -22186.271} C_VEL
LIN {X 0,Y 209.321,Z 532.218,A -85,B 0,C 180,E1 -22188.357,E2 -22188.357} C_VEL
LIN {X 0,Y 210.243,Z 544.7,A -85,B 0,C 180,E1 -22190.57,E2 -22190.57} C_VEL
LIN {X 0,Y 210.243,Z 556.023,A -85,B 0,C 180,E1 -22192.762,E2 -22192.762} C_VEL
LIN {X 0,Y 210.007,Z 558.955,A -85,B 0,C 180,E1 -22193.344,E2 -22193.344} C_VEL
LIN {X 0,Y 206.22,Z 570.848,A -85,B 0,C 180,E1 -22195.488,E2 -22195.488} C_VEL
LIN {X 0,Y 201.998,Z 581.813,A -85,B 0,C 180,E1 -22197.955,E2 -22197.955} C_VEL
LIN {X 0,Y 197.957,Z 591.655,A -85,B 0,C 180,E1 -22200.78,E2 -22200.78} C_VEL
LIN {X 0,Y 193.764,Z 601.038,A -85,B 0,C 180,E1 -22204.199,E2 -22204.199} C_VEL
LIN {X 0,Y 190.697,Z 607.818,A -85,B 0,C 180,E1 -22207.347,E2 -22207.347} C_VEL
LIN {X 0,Y 188.506,Z 613.079,A -85,B 0,C 180,E1 -22210.394,E2 -22210.394} C_VEL
LIN {X 0,Y 185.8,Z 618.794,A -85,B 0,C 180,E1 -22214.646,E2 -22214.646} C_VEL
LIN {X 0,Y 184.194,Z 622.946,A -85,B 0,C 180,E1 -22219.002,E2 -22219.002} C_VEL
LIN {X 0,Y 183.304,Z 625.661,A -85,B 0,C 180,E1 -22223.395,E2 -22223.395} C_VEL
LIN {X 0,Y 183.041,Z 627.018,A -85,B 0,C 180,E1 -22227.8,E2 -22227.8} C_VEL
LIN {X 0,Y 183.068,Z 627.197,A -85,B 0,C 180,E1 -22230,E2 -22230} C_VEL
LIN {X 0,Y 183.081,Z 626.556,A -85,B 0,C 180,E1 -22234.403,E2 -22234.403} C_VEL
LIN {X 0,Y 183.658,Z 624.567,A -85,B 0,C 180,E1 -22238.805,E2 -22238.805} C_VEL
LIN {X 0,Y 184.865,Z 621.192,A -85,B 0,C 180,E1 -22243.185,E2 -22243.185} C_VEL
LIN {X 0,Y 186.972,Z 616.326,A -85,B 0,C 180,E1 -22247.5,E2 -22247.5} C_VEL
LIN {X 0,Y 189.178,Z 611.606,A -85,B 0,C 180,E1 -22250.666,E2 -22250.666} C_VEL
LIN {X 0,Y 192.194,Z 604.766,A -85,B 0,C 180,E1 -22254.292,E2 -22254.292} C_VEL
LIN {X 0,Y 196.043,Z 596.271,A -85,B 0,C 180,E1 -22257.778,E2 -22257.778} C_VEL
LIN {X 0,Y 199.793,Z 587.382,A -85,B 0,C 180,E1 -22260.668,E2 -22260.668} C_VEL
LIN {X 0,Y 204.142,Z 576.615,A -85,B 0,C 180,E1 -22263.424,E2 -22263.424} C_VEL
LIN {X 0,Y 208.166,Z 565.267,A -85,B 0,C 180,E1 -22265.717,E2 -22265.717} C_VEL
LIN {X 0,Y 210.1,Z 559.062,A -85,B 0,C 180,E1 -22266.766,E2 -22266.766} C_VEL
LIN {X 0,Y 210.449,Z 548.812,A -85,B 0,C 180,E1 -22268.798,E2 -22268.798} C_VEL
LIN {X 0,Y 209.807,Z 536.304,A -85,B 0,C 180,E1 -22271.09,E2 -22271.09} C_VEL
LIN {X 0,Y 208.238,Z 524.427,A -85,B 0,C 180,E1 -22273.127,E2 -22273.127} C_VEL
LIN {X 0,Y 205.27,Z 511.252,A -85,B 0,C 180,E1 -22275.341,E2 -22275.341} C_VEL
LIN {X 0,Y 202.724,Z 503.223,A -85,B 0,C 180,E1 -22276.721,E2 -22276.721} C_VEL
LIN {X 0,Y 198.64,Z 495.573,A -85,B 0,C 180,E1 -22278.471,E2 -22278.471} C_VEL
LIN {X 0,Y 196.548,Z 491.752,A -85,B 0,C 180,E1 -22279.372,E2 -22279.372} C_VEL
LIN {X 0,Y 196.354,Z 491.165,A -85,B 0,C 180,E1 -22279.566,E2 -22279.566} C_VEL
LIN {X 0,Y 195.578,Z 485.566,A -85,B 0,C 180,E1 -22283.635,E2 -22283.635} C_VEL
LIN {X 0,Y 194.64,Z 480.399,A -85,B 0,C 180,E1 -22287.798,E2 -22287.798} C_VEL
LIN {X 0,Y 194.497,Z 480.225,A -85,B 0,C 180,E1 -22287.992,E2 -22287.992} C_VEL
LIN {X 0,Y 196.969,Z 489.586,A -85,B 0,C 180,E1 -22290.031,E2 -22290.031} C_VEL
LIN {X 0,Y 194.207,Z 502.87,A -85,B 0,C 180,E1 -22292.814,E2 -22292.814} C_VEL
LIN {X 0,Y 191.821,Z 514.173,A -85,B 0,C 180,E1 -22295.658,E2 -22295.658} C_VEL
LIN {X 0,Y 189.507,Z 524.743,A -85,B 0,C 180,E1 -22298.802,E2 -22298.802} C_VEL
LIN {X 0,Y 187.834,Z 533.881,A -85,B 0,C 180,E1 -22302.02,E2 -22302.02} C_VEL
LIN {X 0,Y 186.22,Z 542.941,A -85,B 0,C 180,E1 -22305.8,E2 -22305.8} C_VEL
LIN {X 0,Y 185.125,Z 551.499,A -85,B 0,C 180,E1 -22310.165,E2 -22310.165} C_VEL
LIN {X 0,Y 184.59,Z 558.483,A -85,B 0,C 180,E1 -22314.538,E2 -22314.538} C_VEL
LIN {X 0,Y 184.3,Z 564.054,A -85,B 0,C 180,E1 -22318.907,E2 -22318.907} C_VEL
LIN {X 0,Y 184.6,Z 567.452,A -85,B 0,C 180,E1 -22322.182,E2 -22322.182} C_VEL
LIN {X 0,Y 185.777,Z 570.915,A -85,B 0,C 180,E1 -22326.516,E2 -22326.516} C_VEL
LIN {X 0,Y 187.732,Z 573.281,A -85,B 0,C 180,E1 -22330.788,E2 -22330.788} C_VEL
LIN {X 0,Y 190.376,Z 574.652,A -85,B 0,C 180,E1 -22334.976,E2 -22334.976} C_VEL
LIN {X 0,Y 193.801,Z 575.064,A -85,B 0,C 180,E1 -22339.049,E2 -22339.049} C_VEL
LIN {X 0,Y 198.208,Z 574.507,A -85,B 0,C 180,E1 -22342.956,E2 -22342.956} C_VEL
LIN {X 0,Y 203.622,Z 572.954,A -85,B 0,C 180,E1 -22346.66,E2 -22346.66} C_VEL
LIN {X 0,Y 209.922,Z 570.478,A -85,B 0,C 180,E1 -22350.145,E2 -22350.145} C_VEL
LIN {X 0,Y 219.042,Z 566.041,A -85,B 0,C 180,E1 -22354.159,E2 -22354.159} C_VEL
LIN {X 0,Y 229.276,Z 560.186,A -85,B 0,C 180,E1 -22357.811,E2 -22357.811} C_VEL
LIN {X 0,Y 240.42,Z 552.85,A -85,B 0,C 180,E1 -22361.011,E2 -22361.011} C_VEL
LIN {X 0,Y 239.629,Z 553.609,A -85,B 0,C 180,E1 -22361.69,E2 -22361.69} C_VEL
LIN {X 0,Y 236.096,Z 556.95,A -85,B 0,C 180,E1 -22363.631,E2 -22363.631} C_VEL
LIN {X 0,Y 231.506,Z 561.431,A -85,B 0,C 180,E1 -22365.715,E2 -22365.715} C_VEL
LIN {X 0,Y 223.356,Z 568.898,A -85,B 0,C 180,E1 -22368.641,E2 -22368.641} C_VEL
LIN {X 0,Y 215.691,Z 575.93,A -85,B 0,C 180,E1 -22371.75,E2 -22371.75} C_VEL
LIN {X 0,Y 206.009,Z 583.987,A -85,B 0,C 180,E1 -22375.743,E2 -22375.743} C_VEL
LIN {X 0,Y 199.525,Z 589.379,A -85,B 0,C 180,E1 -22379.14,E2 -22379.14} C_VEL
LIN {X 0,Y 198.477,Z 591.934,A -85,B 0,C 180,E1 -22379.889,E2 -22379.889} C_VEL
LIN {X 0,Y 196.225,Z 595.832,A -85,B 0,C 180,E1 -22381.005,E2 -22381.005} C_VEL
LIN {X 0,Y 190.999,Z 601.819,A -85,B 0,C 180,E1 -22382.77,E2 -22382.77} C_VEL
LIN {X 0,Y 185.907,Z 607.255,A -85,B 0,C 180,E1 -22384.757,E2 -22384.757} C_VEL
LIN {X 0,Y 183.918,Z 610.277,A -85,B 0,C 180,E1 -22386.2,E2 -22386.2} C_VEL
LIN {X 0,Y 181.298,Z 616.01,A -85,B 0,C 180,E1 -22389.581,E2 -22389.581} C_VEL
LIN {X 0,Y 179.225,Z 620.505,A -85,B 0,C 180,E1 -22392.896,E2 -22392.896} C_VEL
LIN {X 0,Y 177.689,Z 624.024,A -85,B 0,C 180,E1 -22396.272,E2 -22396.272} C_VEL
LIN {X 0,Y 176.47,Z 627.457,A -85,B 0,C 180,E1 -22400.834,E2 -22400.834} C_VEL
LIN {X 0,Y 176.007,Z 629.488,A -85,B 0,C 180,E1 -22405.419,E2 -22405.419} C_VEL
LIN {X 0,Y 176.038,Z 630.159,A -85,B 0,C 180,E1 -22410,E2 -22410} C_VEL
LIN {X 0,Y 176.007,Z 629.471,A -85,B 0,C 180,E1 -22414.581,E2 -22414.581} C_VEL
LIN {X 0,Y 176.462,Z 627.427,A -85,B 0,C 180,E1 -22419.167,E2 -22419.167} C_VEL
LIN {X 0,Y 177.677,Z 623.977,A -85,B 0,C 180,E1 -22423.729,E2 -22423.729} C_VEL
LIN {X 0,Y 179.854,Z 619.019,A -85,B 0,C 180,E1 -22428.217,E2 -22428.217} C_VEL
LIN {X 0,Y 182.054,Z 614.211,A -85,B 0,C 180,E1 -22431.515,E2 -22431.515} C_VEL
LIN {X 0,Y 184.716,Z 608.368,A -85,B 0,C 180,E1 -22434.741,E2 -22434.741} C_VEL
LIN {X 0,Y 188.624,Z 599.97,A -85,B 0,C 180,E1 -22438.363,E2 -22438.363} C_VEL
LIN {X 0,Y 192.525,Z 591.194,A -85,B 0,C 180,E1 -22441.345,E2 -22441.345} C_VEL
LIN {X 0,Y 197.029,Z 580.547,A -85,B 0,C 180,E1 -22444.18,E2 -22444.18} C_VEL
LIN {X 0,Y 200.949,Z 569.761,A -85,B 0,C 180,E1 -22446.481,E2 -22446.481} C_VEL
LIN {X 0,Y 201.731,Z 566.068,A -85,B 0,C 180,E1 -22447.252,E2 -22447.252} C_VEL
LIN {X 0,Y 203.102,Z 553.276,A -85,B 0,C 180,E1 -22449.814,E2 -22449.814} C_VEL
LIN {X 0,Y 203.816,Z 541.811,A -85,B 0,C 180,E1 -22451.761,E2 -22451.761} C_VEL
LIN {X 0,Y 202.875,Z 531.053,A -85,B 0,C 180,E1 -22453.657,E2 -22453.657} C_VEL
LIN {X 0,Y 200.721,Z 519.147,A -85,B 0,C 180,E1 -22455.74,E2 -22455.74} C_VEL
LIN {X 0,Y 197.131,Z 506.529,A -85,B 0,C 180,E1 -22458.015,E2 -22458.015} C_VEL
LIN {X 0,Y 192.698,Z 494.91,A -85,B 0,C 180,E1 -22460.254,E2 -22460.254} C_VEL
LIN {X 0,Y 190.974,Z 490.602,A -85,B 0,C 180,E1 -22461.188,E2 -22461.188} C_VEL
LIN {X 0,Y 190.667,Z 486.708,A -85,B 0,C 180,E1 -22463.204,E2 -22463.204} C_VEL
LIN {X 0,Y 189.374,Z 479.81,A -85,B 0,C 180,E1 -22467.444,E2 -22467.444} C_VEL
LIN {X 0,Y 188.075,Z 473.352,A -85,B 0,C 180,E1 -22472.154,E2 -22472.154} C_VEL
LIN {X 0,Y 187.518,Z 471.299,A -85,B 0,C 180,E1 -22474.092,E2 -22474.092} C_VEL
LIN {X 0,Y 186.079,Z 468.332,A -85,B 0,C 180,E1 -22477.81,E2 -22477.81} C_VEL
LIN {X 0,Y 184.714,Z 465.503,A -85,B 0,C 180,E1 -22482.279,E2 -22482.279} C_VEL
LIN {X 0,Y 183.928,Z 463.396,A -85,B 0,C 180,E1 -22486.746,E2 -22486.746} C_VEL
LIN {X 0,Y 183.447,Z 462.329,A -85,B 0,C 180,E1 -22491.185,E2 -22491.185} C_VEL
LIN {X 0,Y 183.345,Z 461.869,A -85,B 0,C 180,E1 -22497.803,E2 -22497.803} C_VEL
LIN {X 0,Y 183.593,Z 461.979,A -85,B 0,C 180,E1 -22500,E2 -22500} C_VEL
LIN {X 0,Y 183.6,Z 462.495,A -85,B 0,C 180,E1 -22502.194,E2 -22502.194} C_VEL
LIN {X 0,Y 184.093,Z 464.889,A -85,B 0,C 180,E1 -22508.784,E2 -22508.784} C_VEL
LIN {X 0,Y 184.55,Z 467.269,A -85,B 0,C 180,E1 -22513.208,E2 -22513.208} C_VEL
LIN {X 0,Y 185.336,Z 470.239,A -85,B 0,C 180,E1 -22517.66,E2 -22517.66} C_VEL
LIN {X 0,Y 186.2,Z 473.782,A -85,B 0,C 180,E1 -22522.176,E2 -22522.176} C_VEL
LIN {X 0,Y 187.318,Z 477.906,A -85,B 0,C 180,E1 -22526.759,E2 -22526.759} C_VEL
LIN {X 0,Y 188.32,Z 482.906,A -85,B 0,C 180,E1 -22531.498,E2 -22531.498} C_VEL
LIN {X 0,Y 189.254,Z 488.895,A -85,B 0,C 180,E1 -22536.453,E2 -22536.453} C_VEL
LIN {X 0,Y 189.651,Z 491.48,A -85,B 0,C 180,E1 -22538.326,E2 -22538.326} C_VEL
LIN {X 0,Y 191.819,Z 495.494,A -85,B 0,C 180,E1 -22539.369,E2 -22539.369} C_VEL
LIN {X 0,Y 193.147,Z 497.678,A -85,B 0,C 180,E1 -22539.975,E2 -22539.975} C_VEL
LIN {X 0,Y 197.721,Z 506.211,A -85,B 0,C 180,E1 -22542.137,E2 -22542.137} C_VEL
LIN {X 0,Y 199.255,Z 510.541,A -85,B 0,C 180,E1 -22542.996,E2 -22542.996} C_VEL
LIN {X 0,Y 202.023,Z 522.56,A -85,B 0,C 180,E1 -22545.139,E2 -22545.139} C_VEL
LIN {X 0,Y 203.733,Z 534.258,A -85,B 0,C 180,E1 -22547.252,E2 -22547.252} C_VEL
LIN {X 0,Y 204.418,Z 545.983,A -85,B 0,C 180,E1 -22549.447,E2 -22549.447} C_VEL
LIN {X 0,Y 204.237,Z 557.213,A -85,B 0,C 180,E1 -22551.728,E2 -22551.728} C_VEL
LIN {X 0,Y 203.792,Z 560.76,A -85,B 0,C 180,E1 -22552.439,E2 -22552.439} C_VEL
LIN {X 0,Y 199.995,Z 571.966,A -85,B 0,C 180,E1 -22554.562,E2 -22554.562} C_VEL
LIN {X 0,Y 195.989,Z 581.867,A -85,B 0,C 180,E1 -22556.849,E2 -22556.849} C_VEL
LIN {X 0,Y 191.76,Z 591.711,A -85,B 0,C 180,E1 -22559.739,E2 -22559.739} C_VEL
LIN {X 0,Y 187.956,Z 599.879,A -85,B 0,C 180,E1 -22562.739,E2 -22562.739} C_VEL
LIN {X 0,Y 184.269,Z 607.454,A -85,B 0,C 180,E1 -22566.257,E2 -22566.257} C_VEL
LIN {X 0,Y 181.789,Z 613.138,A -85,B 0,C 180,E1 -22569.639,E2 -22569.639} C_VEL
LIN {X 0,Y 178.93,Z 618.853,A -85,B 0,C 180,E1 -22574.041,E2 -22574.041} C_VEL
LIN {X 0,Y 177.206,Z 623.005,A -85,B 0,C 180,E1 -22578.562,E2 -22578.562} C_VEL
LIN {X 0,Y 176.243,Z 625.72,A -85,B 0,C 180,E1 -22583.129,E2 -22583.129} C_VEL
LIN {X 0,Y 175.95,Z 627.077,A -85,B 0,C 180,E1 -22587.711,E2 -22587.711} C_VEL
LIN {X 0,Y 175.982,Z 627.256,A -85,B 0,C 180,E1 -22590,E2 -22590} C_VEL
LIN {X 0,Y 176.013,Z 626.614,A -85,B 0,C 180,E1 -22594.58,E2 -22594.58} C_VEL
LIN {X 0,Y 176.624,Z 624.625,A -85,B 0,C 180,E1 -22599.158,E2 -22599.158} C_VEL
LIN {X 0,Y 177.934,Z 621.249,A -85,B 0,C 180,E1 -22603.709,E2 -22603.709} C_VEL
LIN {X 0,Y 180.177,Z 616.383,A -85,B 0,C 180,E1 -22608.183,E2 -22608.183} C_VEL
LIN {X 0,Y 182.507,Z 611.662,A -85,B 0,C 180,E1 -22611.459,E2 -22611.459} C_VEL
LIN {X 0,Y 185.723,Z 604.82,A -85,B 0,C 180,E1 -22615.196,E2 -22615.196} C_VEL
LIN {X 0,Y 189.774,Z 596.323,A -85,B 0,C 180,E1 -22618.779,E2 -22618.779} C_VEL
LIN {X 0,Y 193.711,Z 587.432,A -85,B 0,C 180,E1 -22621.74,E2 -22621.74} C_VEL
LIN {X 0,Y 198.224,Z 576.662,A -85,B 0,C 180,E1 -22624.561,E2 -22624.561} C_VEL
LIN {X 0,Y 202.207,Z 565.984,A -85,B 0,C 180,E1 -22626.767,E2 -22626.767} C_VEL
LIN {X 0,Y 204.087,Z 560.285,A -85,B 0,C 180,E1 -22627.769,E2 -22627.769} C_VEL
LIN {X 0,Y 204.548,Z 548.848,A -85,B 0,C 180,E1 -22630.14,E2 -22630.14} C_VEL
LIN {X 0,Y 204.085,Z 537.266,A -85,B 0,C 180,E1 -22632.35,E2 -22632.35} C_VEL
LIN {X 0,Y 202.496,Z 524.625,A -85,B 0,C 180,E1 -22634.642,E2 -22634.642} C_VEL
LIN {X 0,Y 199.795,Z 512.396,A -85,B 0,C 180,E1 -22636.833,E2 -22636.833} C_VEL
LIN {X 0,Y 198,Z 506.749,A -85,B 0,C 180,E1 -22637.907,E2 -22637.907} C_VEL
LIN {X 0,Y 194.587,Z 500.24,A -85,B 0,C 180,E1 -22639.534,E2 -22639.534} C_VEL
LIN {X 0,Y 192.23,Z 495.957,A -85,B 0,C 180,E1 -22640.647,E2 -22640.647} C_VEL
LIN {X 0,Y 189.846,Z 491.89,A -85,B 0,C 180,E1 -22641.773,E2 -22641.773} C_VEL
LIN {X 0,Y 189.595,Z 491.237,A -85,B 0,C 180,E1 -22641.955,E2 -22641.955} C_VEL
LIN {X 0,Y 188.835,Z 486.032,A -85,B 0,C 180,E1 -22646.064,E2 -22646.064} C_VEL
LIN {X 0,Y 188.338,Z 483.976,A -85,B 0,C 180,E1 -22647.876,E2 -22647.876} C_VEL
LIN {X 0,Y 188.187,Z 483.83,A -85,B 0,C 180,E1 -22648.162,E2 -22648.162} C_VEL
LIN {X 0,Y 189.762,Z 489.562,A -85,B 0,C 180,E1 -22649.467,E2 -22649.467} C_VEL
LIN {X 0,Y 189.649,Z 492.01,A -85,B 0,C 180,E1 -22649.981,E2 -22649.981} C_VEL
LIN {X 0,Y 186.588,Z 506.115,A -85,B 0,C 180,E1 -22653.128,E2 -22653.128} C_VEL
LIN {X 0,Y 183.809,Z 518.751,A -85,B 0,C 180,E1 -22656.585,E2 -22656.585} C_VEL
LIN {X 0,Y 181.868,Z 528.176,A -85,B 0,C 180,E1 -22659.648,E2 -22659.648} C_VEL
LIN {X 0,Y 179.96,Z 538.196,A -85,B 0,C 180,E1 -22663.552,E2 -22663.552} C_VEL
LIN {X 0,Y 178.45,Z 547.749,A -85,B 0,C 180,E1 -22668.067,E2 -22668.067} C_VEL
LIN {X 0,Y 177.65,Z 554.694,A -85,B 0,C 180,E1 -22672.016,E2 -22672.016} C_VEL
LIN {X 0,Y 177.409,Z 559.723,A -85,B 0,C 180,E1 -22675.456,E2 -22675.456} C_VEL
LIN {X 0,Y 177.214,Z 565.224,A -85,B 0,C 180,E1 -22680,E2 -22680} C_VEL
LIN {X 0,Y 177.967,Z 569.519,A -85,B 0,C 180,E1 -22684.53,E2 -22684.53} C_VEL
LIN {X 0,Y 179.644,Z 572.699,A -85,B 0,C 180,E1 -22689.003,E2 -22689.003} C_VEL
LIN {X 0,Y 182.102,Z 574.855,A -85,B 0,C 180,E1 -22693.389,E2 -22693.389} C_VEL
LIN {X 0,Y 185.305,Z 575.992,A -85,B 0,C 180,E1 -22697.663,E2 -22697.663} C_VEL
LIN {X 0,Y 190.876,Z 576.068,A -85,B 0,C 180,E1 -22703.002,E2 -22703.002} C_VEL
LIN {X 0,Y 197.504,Z 574.732,A -85,B 0,C 180,E1 -22707.554,E2 -22707.554} C_VEL
LIN {X 0,Y 204.099,Z 572.624,A -85,B 0,C 180,E1 -22711.099,E2 -22711.099} C_VEL
LIN {X 0,Y 211.598,Z 569.537,A -85,B 0,C 180,E1 -22714.377,E2 -22714.377} C_VEL
LIN {X 0,Y 222.008,Z 564.473,A -85,B 0,C 180,E1 -22718.119,E2 -22718.119} C_VEL
LIN {X 0,Y 233.322,Z 558.057,A -85,B 0,C 180,E1 -22721.504,E2 -22721.504} C_VEL
LIN {X 0,Y 228.623,Z 562.061,A -85,B 0,C 180,E1 -22723.747,E2 -22723.747} C_VEL
LIN {X 0,Y 224.712,Z 565.447,A -85,B 0,C 180,E1 -22725.275,E2 -22725.275} C_VEL
LIN {X 0,Y 210.252,Z 577.235,A -85,B 0,C 180,E1 -22730.572,E2 -22730.572} C_VEL
LIN {X 0,Y 200.218,Z 584.73,A -85,B 0,C 180,E1 -22734.607,E2 -22734.607} C_VEL
LIN {X 0,Y 193.101,Z 590.139,A -85,B 0,C 180,E1 -22738.301,E2 -22738.301} C_VEL
LIN {X 0,Y 189.296,Z 598.754,A -85,B 0,C 180,E1 -22741.141,E2 -22741.141} C_VEL
LIN {X 0,Y 185.265,Z 607.363,A -85,B 0,C 180,E1 -22744.737,E2 -22744.737} C_VEL
LIN {X 0,Y 183.918,Z 610.277,A -85,B 0,C 180,E1 -22746.2,E2 -22746.2} C_VEL
LIN {X 0,Y 181.994,Z 613.145,A -85,B 0,C 180,E1 -22747.709,E2 -22747.709} C_VEL
LIN {X 0,Y 177.248,Z 617.421,A -85,B 0,C 180,E1 -22750.136,E2 -22750.136} C_VEL
LIN {X 0,Y 172.714,Z 621.088,A -85,B 0,C 180,E1 -22752.775,E2 -22752.775} C_VEL
LIN {X 0,Y 171.181,Z 622.952,A -85,B 0,C 180,E1 -22754.577,E2 -22754.577} C_VEL
LIN {X 0,Y 169.997,Z 625.863,A -85,B 0,C 180,E1 -22758.07,E2 -22758.07} C_VEL
LIN {X 0,Y 169.095,Z 628.585,A -85,B 0,C 180,E1 -22762.837,E2 -22762.837} C_VEL
LIN {X 0,Y 168.865,Z 629.935,A -85,B 0,C 180,E1 -22767.615,E2 -22767.615} C_VEL
LIN {X 0,Y 168.949,Z 630.101,A -85,B 0,C 180,E1 -22770,E2 -22770} C_VEL
LIN {X 0,Y 168.93,Z 629.412,A -85,B 0,C 180,E1 -22774.773,E2 -22774.773} C_VEL
LIN {X 0,Y 169.416,Z 627.368,A -85,B 0,C 180,E1 -22779.552,E2 -22779.552} C_VEL
LIN {X 0,Y 170.73,Z 623.918,A -85,B 0,C 180,E1 -22784.299,E2 -22784.299} C_VEL
LIN {X 0,Y 173.094,Z 618.961,A -85,B 0,C 180,E1 -22788.955,E2 -22788.955} C_VEL
LIN {X 0,Y 176.179,Z 612.454,A -85,B 0,C 180,E1 -22793.437,E2 -22793.437} C_VEL
LIN {X 0,Y 179.944,Z 604.95,A -85,B 0,C 180,E1 -22797.317,E2 -22797.317} C_VEL
LIN {X 0,Y 183.692,Z 597.205,A -85,B 0,C 180,E1 -22800.46,E2 -22800.46} C_VEL
LIN {X 0,Y 187.996,Z 587.853,A -85,B 0,C 180,E1 -22803.464,E2 -22803.464} C_VEL
LIN {X 0,Y 192.592,Z 577.072,A -85,B 0,C 180,E1 -22806.17,E2 -22806.17} C_VEL
LIN {X 0,Y 195.524,Z 568.544,A -85,B 0,C 180,E1 -22807.992,E2 -22807.992} C_VEL
LIN {X 0,Y 197.145,Z 556.391,A -85,B 0,C 180,E1 -22810.592,E2 -22810.592} C_VEL
LIN {X 0,Y 198.211,Z 544.163,A -85,B 0,C 180,E1 -22812.802,E2 -22812.802} C_VEL
LIN {X 0,Y 197.381,Z 532.493,A -85,B 0,C 180,E1 -22814.99,E2 -22814.99} C_VEL
LIN {X 0,Y 195.402,Z 520.874,A -85,B 0,C 180,E1 -22817.156,E2 -22817.156} C_VEL
LIN {X 0,Y 192.295,Z 509.421,A -85,B 0,C 180,E1 -22819.382,E2 -22819.382} C_VEL
LIN {X 0,Y 188.783,Z 499.371,A -85,B 0,C 180,E1 -22821.437,E2 -22821.437} C_VEL
LIN {X 0,Y 186.274,Z 493.682,A -85,B 0,C 180,E1 -22822.774,E2 -22822.774} C_VEL
LIN {X 0,Y 184.918,Z 490.703,A -85,B 0,C 180,E1 -22823.546,E2 -22823.546} C_VEL
LIN {X 0,Y 183.837,Z 484.274,A -85,B 0,C 180,E1 -22827.642,E2 -22827.642} C_VEL
LIN {X 0,Y 182.714,Z 477.834,A -85,B 0,C 180,E1 -22832.511,E2 -22832.511} C_VEL
LIN {X 0,Y 181.945,Z 475.457,A -85,B 0,C 180,E1 -22834.856,E2 -22834.856} C_VEL
LIN {X 0,Y 180.226,Z 471.994,A -85,B 0,C 180,E1 -22839.454,E2 -22839.454} C_VEL
LIN {X 0,Y 179.137,Z 469.414,A -85,B 0,C 180,E1 -22844.06,E2 -22844.06} C_VEL
LIN {X 0,Y 178.389,Z 467.644,A -85,B 0,C 180,E1 -22848.639,E2 -22848.639} C_VEL
LIN {X 0,Y 177.94,Z 466.774,A -85,B 0,C 180,E1 -22853.195,E2 -22853.195} C_VEL
LIN {X 0,Y 178.1,Z 466.495,A -85,B 0,C 180,E1 -22860,E2 -22860} C_VEL
LIN {X 0,Y 177.999,Z 467.731,A -85,B 0,C 180,E1 -22864.529,E2 -22864.529} C_VEL
LIN {X 0,Y 178.505,Z 469.395,A -85,B 0,C 180,E1 -22869.061,E2 -22869.061} C_VEL
LIN {X 0,Y 178.871,Z 471.735,A -85,B 0,C 180,E1 -22873.636,E2 -22873.636} C_VEL
LIN {X 0,Y 179.537,Z 474.66,A -85,B 0,C 180,E1 -22878.25,E2 -22878.25} C_VEL
LIN {X 0,Y 180.43,Z 478.381,A -85,B 0,C 180,E1 -22882.925,E2 -22882.925} C_VEL
LIN {X 0,Y 181.317,Z 481.9,A -85,B 0,C 180,E1 -22886.937,E2 -22886.937} C_VEL
LIN {X 0,Y 182.251,Z 487.1,A -85,B 0,C 180,E1 -22891.965,E2 -22891.965} C_VEL
LIN {X 0,Y 182.875,Z 491.339,A -85,B 0,C 180,E1 -22895.549,E2 -22895.549} C_VEL
LIN {X 0,Y 185.244,Z 495.524,A -85,B 0,C 180,E1 -22896.827,E2 -22896.827} C_VEL
LIN {X 0,Y 186.452,Z 497.418,A -85,B 0,C 180,E1 -22897.442,E2 -22897.442} C_VEL
LIN {X 0,Y 189.946,Z 503.782,A -85,B 0,C 180,E1 -22899.262,E2 -22899.262} C_VEL
LIN {X 0,Y 193.91,Z 511.887,A -85,B 0,C 180,E1 -22901.41,E2 -22901.41} C_VEL
LIN {X 0,Y 196.424,Z 522.928,A -85,B 0,C 180,E1 -22903.533,E2 -22903.533} C_VEL
LIN {X 0,Y 198.257,Z 536.617,A -85,B 0,C 180,E1 -22906.148,E2 -22906.148} C_VEL
LIN {X 0,Y 198.663,Z 547.891,A -85,B 0,C 180,E1 -22908.379,E2 -22908.379} C_VEL
LIN {X 0,Y 198.252,Z 559.259,A -85,B 0,C 180,E1 -22910.82,E2 -22910.82} C_VEL
LIN {X 0,Y 197.666,Z 562.374,A -85,B 0,C 180,E1 -22911.464,E2 -22911.464} C_VEL
LIN {X 0,Y 193.824,Z 573.071,A -85,B 0,C 180,E1 -22913.576,E2 -22913.576} C_VEL
LIN {X 0,Y 189.266,Z 583.678,A -85,B 0,C 180,E1 -22916.152,E2 -22916.152} C_VEL
LIN {X 0,Y 184.96,Z 593.233,A -85,B 0,C 180,E1 -22919.138,E2 -22919.138} C_VEL
LIN {X 0,Y 181.034,Z 601.153,A -85,B 0,C 180,E1 -22922.234,E2 -22922.234} C_VEL
LIN {X 0,Y 177.507,Z 607.991,A -85,B 0,C 180,E1 -22925.594,E2 -22925.594} C_VEL
LIN {X 0,Y 175.106,Z 613.196,A -85,B 0,C 180,E1 -22928.825,E2 -22928.825} C_VEL
LIN {X 0,Y 172.081,Z 618.912,A -85,B 0,C 180,E1 -22933.388,E2 -22933.388} C_VEL
LIN {X 0,Y 170.24,Z 623.064,A -85,B 0,C 180,E1 -22938.088,E2 -22938.088} C_VEL
LIN {X 0,Y 169.176,Z 625.779,A -85,B 0,C 180,E1 -22942.841,E2 -22942.841} C_VEL
LIN {X 0,Y 168.859,Z 627.135,A -85,B 0,C 180,E1 -22947.615,E2 -22947.615} C_VEL
LIN {X 0,Y 168.881,Z 627.314,A -85,B 0,C 180,E1 -22950,E2 -22950} C_VEL
LIN {X 0,Y 168.938,Z 626.672,A -85,B 0,C 180,E1 -22954.773,E2 -22954.773} C_VEL
LIN {X 0,Y 169.612,Z 624.683,A -85,B 0,C 180,E1 -22959.54,E2 -22959.54} C_VEL
LIN {X 0,Y 171.021,Z 621.306,A -85,B 0,C 180,E1 -22964.274,E2 -22964.274} C_VEL
LIN {X 0,Y 172.683,Z 617.837,A -85,B 0,C 180,E1 -22967.773,E2 -22967.773} C_VEL
LIN {X 0,Y 175.035,Z 613.4,A -85,B 0,C 180,E1 -22971.184,E2 -22971.184} C_VEL
LIN {X 0,Y 178.212,Z 607.025,A -85,B 0,C 180,E1 -22975.063,E2 -22975.063} C_VEL
LIN {X 0,Y 182.254,Z 599.026,A -85,B 0,C 180,E1 -22978.817,E2 -22978.817} C_VEL
LIN {X 0,Y 186.245,Z 590.669,A -85,B 0,C 180,E1 -22981.89,E2 -22981.89} C_VEL
LIN {X 0,Y 190.812,Z 580.552,A -85,B 0,C 180,E1 -22984.813,E2 -22984.813} C_VEL
LIN {X 0,Y 195.412,Z 569.227,A -85,B 0,C 180,E1 -22987.366,E2 -22987.366} C_VEL
LIN {X 0,Y 198.136,Z 561.388,A -85,B 0,C 180,E1 -22988.842,E2 -22988.842} C_VEL
LIN {X 0,Y 198.753,Z 550.043,A -85,B 0,C 180,E1 -22991.312,E2 -22991.312} C_VEL
LIN {X 0,Y 198.487,Z 539.231,A -85,B 0,C 180,E1 -22993.49,E2 -22993.49} C_VEL
LIN {X 0,Y 197.087,Z 526.515,A -85,B 0,C 180,E1 -22995.942,E2 -22995.942} C_VEL
LIN {X 0,Y 194.62,Z 514.146,A -85,B 0,C 180,E1 -22998.287,E2 -22998.287} C_VEL
LIN {X 0,Y 193.204,Z 510.145,A -85,B 0,C 180,E1 -22999.189,E2 -22999.189} C_VEL
LIN {X 0,Y 188.673,Z 501.199,A -85,B 0,C 180,E1 -23001.608,E2 -23001.608} C_VEL
LIN {X 0,Y 185.567,Z 495.945,A -85,B 0,C 180,E1 -23003.219,E2 -23003.219} C_VEL
LIN {X 0,Y 183.11,Z 491.833,A -85,B 0,C 180,E1 -23004.528,E2 -23004.528} C_VEL
LIN {X 0,Y 182.889,Z 491.125,A -85,B 0,C 180,E1 -23004.801,E2 -23004.801} C_VEL
LIN {X 0,Y 182.422,Z 488.111,A -85,B 0,C 180,E1 -23007.359,E2 -23007.359} C_VEL
LIN {X 0,Y 181.833,Z 487.311,A -85,B 0,C 180,E1 -23008.291,E2 -23008.291} C_VEL
LIN {X 0,Y 182.861,Z 491.554,A -85,B 0,C 180,E1 -23009.338,E2 -23009.338} C_VEL
LIN {X 0,Y 179.919,Z 504.933,A -85,B 0,C 180,E1 -23012.363,E2 -23012.363} C_VEL
LIN {X 0,Y 177.379,Z 516.263,A -85,B 0,C 180,E1 -23015.475,E2 -23015.475} C_VEL
LIN {X 0,Y 175.112,Z 526.546,A -85,B 0,C 180,E1 -23018.825,E2 -23018.825} C_VEL
LIN {X 0,Y 173.327,Z 535.592,A -85,B 0,C 180,E1 -23022.295,E2 -23022.295} C_VEL
LIN {X 0,Y 171.659,Z 545.808,A -85,B 0,C 180,E1 -23026.986,E2 -23026.986} C_VEL
LIN {X 0,Y 170.748,Z 553.054,A -85,B 0,C 180,E1 -23031.056,E2 -23031.056} C_VEL
LIN {X 0,Y 170.345,Z 559.346,A -85,B 0,C 180,E1 -23035.267,E2 -23035.267} C_VEL
LIN {X 0,Y 170.125,Z 565.123,A -85,B 0,C 180,E1 -23040,E2 -23040} C_VEL
LIN {X 0,Y 170.893,Z 569.687,A -85,B 0,C 180,E1 -23044.718,E2 -23044.718} C_VEL
LIN {X 0,Y 172.647,Z 573.116,A -85,B 0,C 180,E1 -23049.371,E2 -23049.371} C_VEL
LIN {X 0,Y 175.223,Z 575.49,A -85,B 0,C 180,E1 -23053.925,E2 -23053.925} C_VEL
LIN {X 0,Y 178.614,Z 576.912,A -85,B 0,C 180,E1 -23058.347,E2 -23058.347} C_VEL
LIN {X 0,Y 182.925,Z 577.43,A -85,B 0,C 180,E1 -23062.594,E2 -23062.594} C_VEL
LIN {X 0,Y 188.383,Z 576.973,A -85,B 0,C 180,E1 -23066.595,E2 -23066.595} C_VEL
LIN {X 0,Y 194.713,Z 575.649,A -85,B 0,C 180,E1 -23070.352,E2 -23070.352} C_VEL
LIN {X 0,Y 202.135,Z 573.407,A -85,B 0,C 180,E1 -23073.8,E2 -23073.8} C_VEL
LIN {X 0,Y 210.322,Z 570.303,A -85,B 0,C 180,E1 -23076.976,E2 -23076.976} C_VEL
LIN {X 0,Y 221.521,Z 565.177,A -85,B 0,C 180,E1 -23080.571,E2 -23080.571} C_VEL
LIN {X 0,Y 225.207,Z 563.317,A -85,B 0,C 180,E1 -23081.582,E2 -23081.582} C_VEL
LIN {X 0,Y 223.907,Z 564.425,A -85,B 0,C 180,E1 -23082.528,E2 -23082.528} C_VEL
LIN {X 0,Y 219.932,Z 567.466,A -85,B 0,C 180,E1 -23084.028,E2 -23084.028} C_VEL
LIN {X 0,Y 207.225,Z 576.798,A -85,B 0,C 180,E1 -23088.438,E2 -23088.438} C_VEL
LIN {X 0,Y 194.5,Z 585.439,A -85,B 0,C 180,E1 -23093.401,E2 -23093.401} C_VEL
LIN {X 0,Y 186.857,Z 590.494,A -85,B 0,C 180,E1 -23097.271,E2 -23097.271} C_VEL
LIN {X 0,Y 182.44,Z 600.049,A -85,B 0,C 180,E1 -23100.583,E2 -23100.583} C_VEL
LIN {X 0,Y 178.286,Z 608.42,A -85,B 0,C 180,E1 -23104.303,E2 -23104.303} C_VEL
LIN {X 0,Y 175.503,Z 614.243,A -85,B 0,C 180,E1 -23107.64,E2 -23107.64} C_VEL
LIN {X 0,Y 172.432,Z 620.448,A -85,B 0,C 180,E1 -23112.201,E2 -23112.201} C_VEL
LIN {X 0,Y 171.181,Z 622.952,A -85,B 0,C 180,E1 -23114.577,E2 -23114.577} C_VEL
LIN {X 0,Y 169.801,Z 624.657,A -85,B 0,C 180,E1 -23116.429,E2 -23116.429} C_VEL
LIN {X 0,Y 166.046,Z 626.907,A -85,B 0,C 180,E1 -23119.466,E2 -23119.466} C_VEL
LIN {X 0,Y 163.173,Z 628.28,A -85,B 0,C 180,E1 -23122.008,E2 -23122.008} C_VEL
LIN {X 0,Y 161.959,Z 629.055,A -85,B 0,C 180,E1 -23124.034,E2 -23124.034} C_VEL
LIN {X 0,Y 161.854,Z 629.273,A -85,B 0,C 180,E1 -23124.727,E2 -23124.727} C_VEL
LIN {X 0,Y 161.761,Z 629.909,A -85,B 0,C 180,E1 -23127.815,E2 -23127.815} C_VEL
LIN {X 0,Y 161.847,Z 630.042,A -85,B 0,C 180,E1 -23130,E2 -23130} C_VEL
LIN {X 0,Y 161.85,Z 629.354,A -85,B 0,C 180,E1 -23134.982,E2 -23134.982} C_VEL
LIN {X 0,Y 162.394,Z 627.309,A -85,B 0,C 180,E1 -23139.969,E2 -23139.969} C_VEL
LIN {X 0,Y 163.805,Z 623.859,A -85,B 0,C 180,E1 -23144.918,E2 -23144.918} C_VEL
LIN {X 0,Y 166.343,Z 618.902,A -85,B 0,C 180,E1 -23149.755,E2 -23149.755} C_VEL
LIN {X 0,Y 169.43,Z 612.8,A -85,B 0,C 180,E1 -23154.138,E2 -23154.138} C_VEL
LIN {X 0,Y 173.022,Z 606.029,A -85,B 0,C 180,E1 -23157.848,E2 -23157.848} C_VEL
LIN {X 0,Y 176.888,Z 598.508,A -85,B 0,C 180,E1 -23161.098,E2 -23161.098} C_VEL
LIN {X 0,Y 181.289,Z 589.465,A -85,B 0,C 180,E1 -23164.202,E2 -23164.202} C_VEL
LIN {X 0,Y 186.271,Z 578.486,A -85,B 0,C 180,E1 -23167.134,E2 -23167.134} C_VEL
LIN {X 0,Y 189.532,Z 569.658,A -85,B 0,C 180,E1 -23169.078,E2 -23169.078} C_VEL
LIN {X 0,Y 191.526,Z 556.825,A -85,B 0,C 180,E1 -23171.937,E2 -23171.937} C_VEL
LIN {X 0,Y 192.627,Z 546.495,A -85,B 0,C 180,E1 -23173.885,E2 -23173.885} C_VEL
LIN {X 0,Y 192.161,Z 535.927,A -85,B 0,C 180,E1 -23175.981,E2 -23175.981} C_VEL
LIN {X 0,Y 190.565,Z 524.499,A -85,B 0,C 180,E1 -23178.261,E2 -23178.261} C_VEL
LIN {X 0,Y 187.629,Z 512.209,A -85,B 0,C 180,E1 -23180.803,E2 -23180.803} C_VEL
LIN {X 0,Y 184.322,Z 502.371,A -85,B 0,C 180,E1 -23182.986,E2 -23182.986} C_VEL
LIN {X 0,Y 181.61,Z 496.043,A -85,B 0,C 180,E1 -23184.601,E2 -23184.601} C_VEL
LIN {X 0,Y 178.763,Z 491.354,A -85,B 0,C 180,E1 -23186.239,E2 -23186.239} C_VEL
LIN {X 0,Y 178.501,Z 490.583,A -85,B 0,C 180,E1 -23186.55,E2 -23186.55} C_VEL
LIN {X 0,Y 177.567,Z 485.081,A -85,B 0,C 180,E1 -23190.546,E2 -23190.546} C_VEL
LIN {X 0,Y 176.945,Z 480.889,A -85,B 0,C 180,E1 -23194.094,E2 -23194.094} C_VEL
LIN {X 0,Y 175.186,Z 477.24,A -85,B 0,C 180,E1 -23198.835,E2 -23198.835} C_VEL
LIN {X 0,Y 173.936,Z 474.438,A -85,B 0,C 180,E1 -23203.57,E2 -23203.57} C_VEL
LIN {X 0,Y 173.385,Z 472.99,A -85,B 0,C 180,E1 -23206.611,E2 -23206.611} C_VEL
LIN {X 0,Y 172.869,Z 471.868,A -85,B 0,C 180,E1 -23210.641,E2 -23210.641} C_VEL
LIN {X 0,Y 172.511,Z 471.072,A -85,B 0,C 180,E1 -23217.665,E2 -23217.665} C_VEL
LIN {X 0,Y 172.684,Z 471.107,A -85,B 0,C 180,E1 -23220,E2 -23220} C_VEL
LIN {X 0,Y 172.516,Z 472.273,A -85,B 0,C 180,E1 -23224.674,E2 -23224.674} C_VEL
LIN {X 0,Y 172.874,Z 473.878,A -85,B 0,C 180,E1 -23229.359,E2 -23229.359} C_VEL
LIN {X 0,Y 173.199,Z 476.273,A -85,B 0,C 180,E1 -23234.091,E2 -23234.091} C_VEL
LIN {X 0,Y 173.843,Z 479.314,A -85,B 0,C 180,E1 -23238.87,E2 -23238.87} C_VEL
LIN {X 0,Y 174.952,Z 483.992,A -85,B 0,C 180,E1 -23244.948,E2 -23244.948} C_VEL
LIN {X 0,Y 175.819,Z 488.723,A -85,B 0,C 180,E1 -23249.978,E2 -23249.978} C_VEL
LIN {X 0,Y 176.28,Z 491.507,A -85,B 0,C 180,E1 -23252.448,E2 -23252.448} C_VEL
LIN {X 0,Y 178.886,Z 495.894,A -85,B 0,C 180,E1 -23254.046,E2 -23254.046} C_VEL
LIN {X 0,Y 180.381,Z 498.234,A -85,B 0,C 180,E1 -23254.908,E2 -23254.908} C_VEL
LIN {X 0,Y 183.288,Z 503.379,A -85,B 0,C 180,E1 -23256.611,E2 -23256.611} C_VEL
LIN {X 0,Y 187.648,Z 511.882,A -85,B 0,C 180,E1 -23259.19,E2 -23259.19} C_VEL
LIN {X 0,Y 189.826,Z 517.474,A -85,B 0,C 180,E1 -23260.646,E2 -23260.646} C_VEL
LIN {X 0,Y 192.003,Z 530.536,A -85,B 0,C 180,E1 -23263.268,E2 -23263.268} C_VEL
LIN {X 0,Y 192.981,Z 542.458,A -85,B 0,C 180,E1 -23265.722,E2 -23265.722} C_VEL
LIN {X 0,Y 192.822,Z 554.208,A -85,B 0,C 180,E1 -23268.234,E2 -23268.234} C_VEL
LIN {X 0,Y 192.235,Z 561.619,A -85,B 0,C 180,E1 -23269.946,E2 -23269.946} C_VEL
LIN {X 0,Y 189.501,Z 569.855,A -85,B 0,C 180,E1 -23271.596,E2 -23271.596} C_VEL
LIN {X 0,Y 185.127,Z 580.125,A -85,B 0,C 180,E1 -23273.954,E2 -23273.954} C_VEL
LIN {X 0,Y 181.086,Z 588.74,A -85,B 0,C 180,E1 -23276.424,E2 -23276.424} C_VEL
LIN {X 0,Y 176.8,Z 597.432,A -85,B 0,C 180,E1 -23279.547,E2 -23279.547} C_VEL
LIN {X 0,Y 172.308,Z 605.758,A -85,B 0,C 180,E1 -23283.342,E2 -23283.342} C_VEL
LIN {X 0,Y 169.299,Z 611.549,A -85,B 0,C 180,E1 -23286.773,E2 -23286.773} C_VEL
LIN {X 0,Y 166.759,Z 616.317,A -85,B 0,C 180,E1 -23290.296,E2 -23290.296} C_VEL
LIN {X 0,Y 164.156,Z 621.234,A -85,B 0,C 180,E1 -23295.115,E2 -23295.115} C_VEL
LIN {X 0,Y 162.595,Z 624.654,A -85,B 0,C 180,E1 -23300.044,E2 -23300.044} C_VEL
LIN {X 0,Y 161.859,Z 626.682,A -85,B 0,C 180,E1 -23305.018,E2 -23305.018} C_VEL
LIN {X 0,Y 161.78,Z 627.373,A -85,B 0,C 180,E1 -23310,E2 -23310} C_VEL
LIN {X 0,Y 161.858,Z 626.73,A -85,B 0,C 180,E1 -23314.982,E2 -23314.982} C_VEL
LIN {X 0,Y 162.592,Z 624.741,A -85,B 0,C 180,E1 -23319.956,E2 -23319.956} C_VEL
LIN {X 0,Y 164.11,Z 621.364,A -85,B 0,C 180,E1 -23324.889,E2 -23324.889} C_VEL
LIN {X 0,Y 165.916,Z 617.894,A -85,B 0,C 180,E1 -23328.523,E2 -23328.523} C_VEL
LIN {X 0,Y 168.386,Z 613.456,A -85,B 0,C 180,E1 -23332.064,E2 -23332.064} C_VEL
LIN {X 0,Y 171.411,Z 607.741,A -85,B 0,C 180,E1 -23335.697,E2 -23335.697} C_VEL
LIN {X 0,Y 175.377,Z 600.295,A -85,B 0,C 180,E1 -23339.4,E2 -23339.4} C_VEL
LIN {X 0,Y 179.496,Z 592.187,A -85,B 0,C 180,E1 -23342.573,E2 -23342.573} C_VEL
LIN {X 0,Y 184.173,Z 582.409,A -85,B 0,C 180,E1 -23345.587,E2 -23345.587} C_VEL
LIN {X 0,Y 188.945,Z 571.537,A -85,B 0,C 180,E1 -23348.198,E2 -23348.198} C_VEL
LIN {X 0,Y 192.287,Z 562.071,A -85,B 0,C 180,E1 -23350.087,E2 -23350.087} C_VEL
LIN {X 0,Y 193.07,Z 550.08,A -85,B 0,C 180,E1 -23352.811,E2 -23352.811} C_VEL
LIN {X 0,Y 192.791,Z 537.914,A -85,B 0,C 180,E1 -23355.376,E2 -23355.376} C_VEL
LIN {X 0,Y 191.634,Z 527.168,A -85,B 0,C 180,E1 -23357.555,E2 -23357.555} C_VEL
LIN {X 0,Y 189.529,Z 516.203,A -85,B 0,C 180,E1 -23359.8,E2 -23359.8} C_VEL
LIN {X 0,Y 186.158,Z 508.806,A -85,B 0,C 180,E1 -23361.9,E2 -23361.9} C_VEL
LIN {X 0,Y 184.459,Z 505.461,A -85,B 0,C 180,E1 -23362.925,E2 -23362.925} C_VEL
LIN {X 0,Y 181.966,Z 501.003,A -85,B 0,C 180,E1 -23364.366,E2 -23364.366} C_VEL
LIN {X 0,Y 179.286,Z 496.354,A -85,B 0,C 180,E1 -23365.956,E2 -23365.956} C_VEL
LIN {X 0,Y 175.887,Z 491.29,A -85,B 0,C 180,E1 -23368.005,E2 -23368.005} C_VEL
LIN {X 0,Y 175.485,Z 490.958,A -85,B 0,C 180,E1 -23368.591,E2 -23368.591} C_VEL
LIN {X 0,Y 175.792,Z 492.7,A -85,B 0,C 180,E1 -23369.02,E2 -23369.02} C_VEL
LIN {X 0,Y 172.529,Z 506.815,A -85,B 0,C 180,E1 -23372.395,E2 -23372.395} C_VEL
LIN {X 0,Y 170.001,Z 517.805,A -85,B 0,C 180,E1 -23375.581,E2 -23375.581} C_VEL
LIN {X 0,Y 167.515,Z 529.804,A -85,B 0,C 180,E1 -23379.749,E2 -23379.749} C_VEL
LIN {X 0,Y 165.504,Z 539.784,A -85,B 0,C 180,E1 -23383.977,E2 -23383.977} C_VEL
LIN {X 0,Y 164.078,Z 549.301,A -85,B 0,C 180,E1 -23388.886,E2 -23388.886} C_VEL
LIN {X 0,Y 163.346,Z 557.164,A -85,B 0,C 180,E1 -23393.825,E2 -23393.825} C_VEL
LIN {X 0,Y 163.037,Z 563.5,A -85,B 0,C 180,E1 -23398.765,E2 -23398.765} C_VEL
LIN {X 0,Y 163.538,Z 568.631,A -85,B 0,C 180,E1 -23403.696,E2 -23403.696} C_VEL
LIN {X 0,Y 165.65,Z 573.392,A -85,B 0,C 180,E1 -23409.771,E2 -23409.771} C_VEL
LIN {X 0,Y 168.358,Z 576.08,A -85,B 0,C 180,E1 -23414.505,E2 -23414.505} C_VEL
LIN {X 0,Y 171.932,Z 577.803,A -85,B 0,C 180,E1 -23419.087,E2 -23419.087} C_VEL
LIN {X 0,Y 176.478,Z 578.562,A -85,B 0,C 180,E1 -23423.468,E2 -23423.468} C_VEL
LIN {X 0,Y 182.206,Z 578.434,A -85,B 0,C 180,E1 -23427.572,E2 -23427.572} C_VEL
LIN {X 0,Y 188.831,Z 577.474,A -85,B 0,C 180,E1 -23431.403,E2 -23431.403} C_VEL
LIN {X 0,Y 196.546,Z 575.55,A -85,B 0,C 180,E1 -23434.898,E2 -23434.898} C_VEL
LIN {X 0,Y 205.032,Z 572.817,A -85,B 0,C 180,E1 -23438.097,E2 -23438.097} C_VEL
LIN {X 0,Y 217.411,Z 567.906,A -85,B 0,C 180,E1 -23441.97,E2 -23441.97} C_VEL
LIN {X 0,Y 212.897,Z 570.929,A -85,B 0,C 180,E1 -23443.427,E2 -23443.427} C_VEL
LIN {X 0,Y 199.655,Z 579.604,A -85,B 0,C 180,E1 -23448.024,E2 -23448.024} C_VEL
LIN {X 0,Y 188.879,Z 586.008,A -85,B 0,C 180,E1 -23452.124,E2 -23452.124} C_VEL
LIN {X 0,Y 180.712,Z 590.848,A -85,B 0,C 180,E1 -23456.177,E2 -23456.177} C_VEL
LIN {X 0,Y 176.264,Z 599.997,A -85,B 0,C 180,E1 -23459.445,E2 -23459.445} C_VEL
LIN {X 0,Y 171.869,Z 608.366,A -85,B 0,C 180,E1 -23463.269,E2 -23463.269} C_VEL
LIN {X 0,Y 168.885,Z 614.247,A -85,B 0,C 180,E1 -23466.756,E2 -23466.756} C_VEL
LIN {X 0,Y 165.639,Z 620.391,A -85,B 0,C 180,E1 -23471.445,E2 -23471.445} C_VEL
LIN {X 0,Y 163.817,Z 623.909,A -85,B 0,C 180,E1 -23475.084,E2 -23475.084} C_VEL
LIN {X 0,Y 162.402,Z 627.341,A -85,B 0,C 180,E1 -23480.032,E2 -23480.032} C_VEL
LIN {X 0,Y 161.854,Z 629.273,A -85,B 0,C 180,E1 -23484.727,E2 -23484.727} C_VEL
LIN {X 0,Y 161.141,Z 629.827,A -85,B 0,C 180,E1 -23486.795,E2 -23486.795} C_VEL
LIN {X 0,Y 159.52,Z 630.091,A -85,B 0,C 180,E1 -23488.839,E2 -23488.839} C_VEL
LIN {X 0,Y 155.8,Z 629.81,A -85,B 0,C 180,E1 -23493.003,E2 -23493.003} C_VEL
LIN {X 0,Y 154.825,Z 629.303,A -85,B 0,C 180,E1 -23495.184,E2 -23495.184} C_VEL
LIN {X 0,Y 154.778,Z 629.063,A -85,B 0,C 180,E1 -23495.921,E2 -23495.921} C_VEL
LIN {X 0,Y 155.392,Z 627.25,A -85,B 0,C 180,E1 -23500.423,E2 -23500.423} C_VEL
LIN {X 0,Y 156.907,Z 623.8,A -85,B 0,C 180,E1 -23505.59,E2 -23505.59} C_VEL
LIN {X 0,Y 159.617,Z 618.843,A -85,B 0,C 180,E1 -23510.625,E2 -23510.625} C_VEL
LIN {X 0,Y 162.658,Z 613.207,A -85,B 0,C 180,E1 -23514.859,E2 -23514.859} C_VEL
LIN {X 0,Y 166.737,Z 605.971,A -85,B 0,C 180,E1 -23518.995,E2 -23518.995} C_VEL
LIN {X 0,Y 171.523,Z 597.092,A -85,B 0,C 180,E1 -23522.882,E2 -23522.882} C_VEL
LIN {X 0,Y 176.298,Z 587.744,A -85,B 0,C 180,E1 -23526.015,E2 -23526.015} C_VEL
LIN {X 0,Y 181.401,Z 576.582,A -85,B 0,C 180,E1 -23528.929,E2 -23528.929} C_VEL
LIN {X 0,Y 183.551,Z 571.068,A -85,B 0,C 180,E1 -23530.159,E2 -23530.159} C_VEL
LIN {X 0,Y 185.674,Z 559.194,A -85,B 0,C 180,E1 -23532.947,E2 -23532.947} C_VEL
LIN {X 0,Y 187.102,Z 547.755,A -85,B 0,C 180,E1 -23535.25,E2 -23535.25} C_VEL
LIN {X 0,Y 186.827,Z 537.675,A -85,B 0,C 180,E1 -23537.381,E2 -23537.381} C_VEL
LIN {X 0,Y 185.662,Z 527.723,A -85,B 0,C 180,E1 -23539.492,E2 -23539.492} C_VEL
LIN {X 0,Y 183.381,Z 516.694,A -85,B 0,C 180,E1 -23541.918,E2 -23541.918} C_VEL
LIN {X 0,Y 180.573,Z 507.008,A -85,B 0,C 180,E1 -23544.196,E2 -23544.196} C_VEL
LIN {X 0,Y 178.284,Z 501.305,A -85,B 0,C 180,E1 -23545.739,E2 -23545.739} C_VEL
LIN {X 0,Y 174.067,Z 494.13,A -85,B 0,C 180,E1 -23548.417,E2 -23548.417} C_VEL
LIN {X 0,Y 172.233,Z 490.774,A -85,B 0,C 180,E1 -23549.74,E2 -23549.74} C_VEL
LIN {X 0,Y 171.478,Z 485.322,A -85,B 0,C 180,E1 -23554.378,E2 -23554.378} C_VEL
LIN {X 0,Y 170.081,Z 482.431,A -85,B 0,C 180,E1 -23558.168,E2 -23558.168} C_VEL
LIN {X 0,Y 168.658,Z 479.258,A -85,B 0,C 180,E1 -23563.419,E2 -23563.419} C_VEL
LIN {X 0,Y 167.901,Z 477.321,A -85,B 0,C 180,E1 -23567.919,E2 -23567.919} C_VEL
LIN {X 0,Y 167.276,Z 476.178,A -85,B 0,C 180,E1 -23572.759,E2 -23572.759} C_VEL
LIN {X 0,Y 167.098,Z 475.672,A -85,B 0,C 180,E1 -23577.59,E2 -23577.59} C_VEL
LIN {X 0,Y 167.202,Z 475.642,A -85,B 0,C 180,E1 -23580,E2 -23580} C_VEL
LIN {X 0,Y 166.959,Z 476.763,A -85,B 0,C 180,E1 -23584.83,E2 -23584.83} C_VEL
LIN {X 0,Y 167.27,Z 478.403,A -85,B 0,C 180,E1 -23589.675,E2 -23589.675} C_VEL
LIN {X 0,Y 167.596,Z 481.209,A -85,B 0,C 180,E1 -23595.315,E2 -23595.315} C_VEL
LIN {X 0,Y 168.084,Z 483.92,A -85,B 0,C 180,E1 -23599.542,E2 -23599.542} C_VEL
LIN {X 0,Y 168.95,Z 487.621,A -85,B 0,C 180,E1 -23604.581,E2 -23604.581} C_VEL
LIN {X 0,Y 169.695,Z 491.515,A -85,B 0,C 180,E1 -23608.77,E2 -23608.77} C_VEL
LIN {X 0,Y 172.4,Z 495.95,A -85,B 0,C 180,E1 -23610.72,E2 -23610.72} C_VEL
LIN {X 0,Y 173.774,Z 497.956,A -85,B 0,C 180,E1 -23611.635,E2 -23611.635} C_VEL
LIN {X 0,Y 177.185,Z 503.773,A -85,B 0,C 180,E1 -23613.903,E2 -23613.903} C_VEL
LIN {X 0,Y 179.803,Z 508.816,A -85,B 0,C 180,E1 -23615.66,E2 -23615.66} C_VEL
LIN {X 0,Y 183.466,Z 516.503,A -85,B 0,C 180,E1 -23618.149,E2 -23618.149} C_VEL
LIN {X 0,Y 185.165,Z 521.233,A -85,B 0,C 180,E1 -23619.476,E2 -23619.476} C_VEL
LIN {X 0,Y 186.727,Z 531.907,A -85,B 0,C 180,E1 -23621.764,E2 -23621.764} C_VEL
LIN {X 0,Y 187.465,Z 543.789,A -85,B 0,C 180,E1 -23624.333,E2 -23624.333} C_VEL
LIN {X 0,Y 187.169,Z 554.819,A -85,B 0,C 180,E1 -23626.809,E2 -23626.809} C_VEL
LIN {X 0,Y 186.359,Z 563.113,A -85,B 0,C 180,E1 -23628.82,E2 -23628.82} C_VEL
LIN {X 0,Y 183.527,Z 571.055,A -85,B 0,C 180,E1 -23630.458,E2 -23630.458} C_VEL
LIN {X 0,Y 178.534,Z 582.03,A -85,B 0,C 180,E1 -23633.107,E2 -23633.107} C_VEL
LIN {X 0,Y 173.642,Z 591.88,A -85,B 0,C 180,E1 -23636.185,E2 -23636.185} C_VEL
LIN {X 0,Y 169.252,Z 600.051,A -85,B 0,C 180,E1 -23639.425,E2 -23639.425} C_VEL
LIN {X 0,Y 164.669,Z 608.053,A -85,B 0,C 180,E1 -23643.513,E2 -23643.513} C_VEL
LIN {X 0,Y 160.959,Z 614.908,A -85,B 0,C 180,E1 -23648.214,E2 -23648.214} C_VEL
LIN {X 0,Y 157.85,Z 620.24,A -85,B 0,C 180,E1 -23653.178,E2 -23653.178} C_VEL
LIN {X 0,Y 156.314,Z 623.183,A -85,B 0,C 180,E1 -23657.009,E2 -23657.009} C_VEL
LIN {X 0,Y 155.074,Z 625.897,A -85,B 0,C 180,E1 -23662.186,E2 -23662.186} C_VEL
LIN {X 0,Y 154.667,Z 627.253,A -85,B 0,C 180,E1 -23667.396,E2 -23667.396} C_VEL
LIN {X 0,Y 154.657,Z 627.365,A -85,B 0,C 180,E1 -23671.301,E2 -23671.301} C_VEL
LIN {X 0,Y 154.771,Z 626.789,A -85,B 0,C 180,E1 -23675.211,E2 -23675.211} C_VEL
LIN {X 0,Y 155.593,Z 624.798,A -85,B 0,C 180,E1 -23680.409,E2 -23680.409} C_VEL
LIN {X 0,Y 157.231,Z 621.421,A -85,B 0,C 180,E1 -23685.557,E2 -23685.557} C_VEL
LIN {X 0,Y 159.185,Z 617.95,A -85,B 0,C 180,E1 -23689.337,E2 -23689.337} C_VEL
LIN {X 0,Y 161.784,Z 613.512,A -85,B 0,C 180,E1 -23693.015,E2 -23693.015} C_VEL
LIN {X 0,Y 164.882,Z 608.025,A -85,B 0,C 180,E1 -23696.637,E2 -23696.637} C_VEL
LIN {X 0,Y 169.209,Z 600.348,A -85,B 0,C 180,E1 -23700.584,E2 -23700.584} C_VEL
LIN {X 0,Y 173.544,Z 592.238,A -85,B 0,C 180,E1 -23703.837,E2 -23703.837} C_VEL
LIN {X 0,Y 178.447,Z 582.458,A -85,B 0,C 180,E1 -23706.914,E2 -23706.914} C_VEL
LIN {X 0,Y 183.412,Z 571.582,A -85,B 0,C 180,E1 -23709.571,E2 -23709.571} C_VEL
LIN {X 0,Y 186.363,Z 563.815,A -85,B 0,C 180,E1 -23711.154,E2 -23711.154} C_VEL
LIN {X 0,Y 187.448,Z 551.668,A -85,B 0,C 180,E1 -23714.049,E2 -23714.049} C_VEL
LIN {X 0,Y 187.41,Z 540.301,A -85,B 0,C 180,E1 -23716.59,E2 -23716.59} C_VEL
LIN {X 0,Y 186.449,Z 528.874,A -85,B 0,C 180,E1 -23719.05,E2 -23719.05} C_VEL
LIN {X 0,Y 184.927,Z 520.03,A -85,B 0,C 180,E1 -23720.991,E2 -23720.991} C_VEL
LIN {X 0,Y 181.087,Z 511.196,A -85,B 0,C 180,E1 -23723.73,E2 -23723.73} C_VEL
LIN {X 0,Y 178.309,Z 505.876,A -85,B 0,C 180,E1 -23725.573,E2 -23725.573} C_VEL
LIN {X 0,Y 176.032,Z 501.714,A -85,B 0,C 180,E1 -23727.081,E2 -23727.081} C_VEL
LIN {X 0,Y 174.89,Z 499.993,A -85,B 0,C 180,E1 -23727.828,E2 -23727.828} C_VEL
LIN {X 0,Y 170.881,Z 505.808,A -85,B 0,C 180,E1 -23729.397,E2 -23729.397} C_VEL
LIN {X 0,Y 167.668,Z 509.062,A -85,B 0,C 180,E1 -23730.838,E2 -23730.838} C_VEL
LIN {X 0,Y 166.255,Z 509.859,A -85,B 0,C 180,E1 -23731.604,E2 -23731.604} C_VEL
LIN {X 0,Y 165.274,Z 509.448,A -85,B 0,C 180,E1 -23732.3,E2 -23732.3} C_VEL
LIN {X 0,Y 165.157,Z 508.847,A -85,B 0,C 180,E1 -23732.468,E2 -23732.468} C_VEL
LIN {X 0,Y 162.08,Z 521.374,A -85,B 0,C 180,E1 -23736.404,E2 -23736.404} C_VEL
LIN {X 0,Y 159.786,Z 532.693,A -85,B 0,C 180,E1 -23740.738,E2 -23740.738} C_VEL
LIN {X 0,Y 157.936,Z 542.345,A -85,B 0,C 180,E1 -23745.175,E2 -23745.175} C_VEL
LIN {X 0,Y 156.828,Z 550.545,A -85,B 0,C 180,E1 -23749.673,E2 -23749.673} C_VEL
LIN {X 0,Y 156.218,Z 558.262,A -85,B 0,C 180,E1 -23754.838,E2 -23754.838} C_VEL
LIN {X 0,Y 155.954,Z 564.584,A -85,B 0,C 180,E1 -23760,E2 -23760} C_VEL
LIN {X 0,Y 156.76,Z 569.656,A -85,B 0,C 180,E1 -23765.144,E2 -23765.144} C_VEL
LIN {X 0,Y 158.665,Z 573.652,A -85,B 0,C 180,E1 -23770.205,E2 -23770.205} C_VEL
LIN {X 0,Y 161.507,Z 576.557,A -85,B 0,C 180,E1 -23775.135,E2 -23775.135} C_VEL
LIN {X 0,Y 165.268,Z 578.543,A -85,B 0,C 180,E1 -23779.889,E2 -23779.889} C_VEL
LIN {X 0,Y 170.073,Z 579.656,A -85,B 0,C 180,E1 -23784.408,E2 -23784.408} C_VEL
LIN {X 0,Y 176.074,Z 579.825,A -85,B 0,C 180,E1 -23788.619,E2 -23788.619} C_VEL
LIN {X 0,Y 182.982,Z 579.168,A -85,B 0,C 180,E1 -23792.528,E2 -23792.528} C_VEL
LIN {X 0,Y 191.033,Z 577.651,A -85,B 0,C 180,E1 -23796.06,E2 -23796.06} C_VEL
LIN {X 0,Y 199.821,Z 575.286,A -85,B 0,C 180,E1 -23799.278,E2 -23799.278} C_VEL
LIN {X 0,Y 204.474,Z 573.813,A -85,B 0,C 180,E1 -23800.772,E2 -23800.772} C_VEL
LIN {X 0,Y 208.215,Z 572.577,A -85,B 0,C 180,E1 -23802.048,E2 -23802.048} C_VEL
LIN {X 0,Y 192.161,Z 581.897,A -85,B 0,C 180,E1 -23807.421,E2 -23807.421} C_VEL
LIN {X 0,Y 181.298,Z 587.553,A -85,B 0,C 180,E1 -23811.666,E2 -23811.666} C_VEL
LIN {X 0,Y 174.841,Z 590.798,A -85,B 0,C 180,E1 -23814.878,E2 -23814.878} C_VEL
LIN {X 0,Y 170.153,Z 599.945,A -85,B 0,C 180,E1 -23818.222,E2 -23818.222} C_VEL
LIN {X 0,Y 165.534,Z 608.312,A -85,B 0,C 180,E1 -23822.159,E2 -23822.159} C_VEL
LIN {X 0,Y 162.007,Z 614.807,A -85,B 0,C 180,E1 -23826.171,E2 -23826.171} C_VEL
LIN {X 0,Y 158.887,Z 620.335,A -85,B 0,C 180,E1 -23830.625,E2 -23830.625} C_VEL
LIN {X 0,Y 156.919,Z 623.852,A -85,B 0,C 180,E1 -23834.412,E2 -23834.412} C_VEL
LIN {X 0,Y 155.4,Z 627.283,A -85,B 0,C 180,E1 -23839.578,E2 -23839.578} C_VEL
LIN {X 0,Y 154.753,Z 629.314,A -85,B 0,C 180,E1 -23844.789,E2 -23844.789} C_VEL
LIN {X 0,Y 154.744,Z 629.984,A -85,B 0,C 180,E1 -23850,E2 -23850} C_VEL
LIN {X 0,Y 154.753,Z 629.295,A -85,B 0,C 180,E1 -23855.211,E2 -23855.211} C_VEL
LIN {X 0,Y 154.778,Z 629.063,A -85,B 0,C 180,E1 -23855.921,E2 -23855.921} C_VEL
LIN {X 0,Y 154.29,Z 628.346,A -85,B 0,C 180,E1 -23858.084,E2 -23858.084} C_VEL
LIN {X 0,Y 152.037,Z 626.686,A -85,B 0,C 180,E1 -23861.648,E2 -23861.648} C_VEL
LIN {X 0,Y 150.459,Z 624.987,A -85,B 0,C 180,E1 -23864.541,E2 -23864.541} C_VEL
LIN {X 0,Y 150.307,Z 623.417,A -85,B 0,C 180,E1 -23866.724,E2 -23866.724} C_VEL
LIN {X 0,Y 150.57,Z 622.844,A -85,B 0,C 180,E1 -23867.441,E2 -23867.441} C_VEL
LIN {X 0,Y 152.935,Z 618.784,A -85,B 0,C 180,E1 -23871.57,E2 -23871.57} C_VEL
LIN {X 0,Y 155.912,Z 613.618,A -85,B 0,C 180,E1 -23875.64,E2 -23875.64} C_VEL
LIN {X 0,Y 159.873,Z 607.025,A -85,B 0,C 180,E1 -23879.64,E2 -23879.64} C_VEL
LIN {X 0,Y 164.819,Z 598.395,A -85,B 0,C 180,E1 -23883.665,E2 -23883.665} C_VEL
LIN {X 0,Y 169.722,Z 589.355,A -85,B 0,C 180,E1 -23886.901,E2 -23886.901} C_VEL
LIN {X 0,Y 175.105,Z 578.38,A -85,B 0,C 180,E1 -23889.954,E2 -23889.954} C_VEL
LIN {X 0,Y 177.369,Z 573.175,A -85,B 0,C 180,E1 -23891.163,E2 -23891.163} C_VEL
LIN {X 0,Y 179.799,Z 561.974,A -85,B 0,C 180,E1 -23893.933,E2 -23893.933} C_VEL
LIN {X 0,Y 181.629,Z 550.741,A -85,B 0,C 180,E1 -23896.318,E2 -23896.318} C_VEL
LIN {X 0,Y 181.677,Z 541.351,A -85,B 0,C 180,E1 -23898.409,E2 -23898.409} C_VEL
LIN {X 0,Y 180.91,Z 531.644,A -85,B 0,C 180,E1 -23900.604,E2 -23900.604} C_VEL
LIN {X 0,Y 179.063,Z 520.762,A -85,B 0,C 180,E1 -23903.147,E2 -23903.147} C_VEL
LIN {X 0,Y 176.456,Z 510.578,A -85,B 0,C 180,E1 -23905.68,E2 -23905.68} C_VEL
LIN {X 0,Y 174.679,Z 506.103,A -85,B 0,C 180,E1 -23907.07,E2 -23907.07} C_VEL
LIN {X 0,Y 171.26,Z 499.755,A -85,B 0,C 180,E1 -23909.517,E2 -23909.517} C_VEL
LIN {X 0,Y 169.013,Z 495.895,A -85,B 0,C 180,E1 -23911.178,E2 -23911.178} C_VEL
LIN {X 0,Y 166.152,Z 490.958,A -85,B 0,C 180,E1 -23913.494,E2 -23913.494} C_VEL
LIN {X 0,Y 165.847,Z 489.488,A -85,B 0,C 180,E1 -23914.928,E2 -23914.928} C_VEL
LIN {X 0,Y 163.987,Z 485.577,A -85,B 0,C 180,E1 -23920.537,E2 -23920.537} C_VEL
LIN {X 0,Y 163.022,Z 483.187,A -85,B 0,C 180,E1 -23925.009,E2 -23925.009} C_VEL
LIN {X 0,Y 162.249,Z 481.384,A -85,B 0,C 180,E1 -23930.023,E2 -23930.023} C_VEL
LIN {X 0,Y 161.701,Z 480.52,A -85,B 0,C 180,E1 -23935.013,E2 -23935.013} C_VEL
LIN {X 0,Y 161.757,Z 480.226,A -85,B 0,C 180,E1 -23940,E2 -23940} C_VEL
LIN {X 0,Y 161.439,Z 481.304,A -85,B 0,C 180,E1 -23944.995,E2 -23944.995} C_VEL
LIN {X 0,Y 161.656,Z 482.913,A -85,B 0,C 180,E1 -23950.015,E2 -23950.015} C_VEL
LIN {X 0,Y 161.85,Z 485.326,A -85,B 0,C 180,E1 -23955.102,E2 -23955.102} C_VEL
LIN {X 0,Y 162.35,Z 488.541,A -85,B 0,C 180,E1 -23960.262,E2 -23960.262} C_VEL
LIN {X 0,Y 163.048,Z 491.402,A -85,B 0,C 180,E1 -23964.174,E2 -23964.174} C_VEL
LIN {X 0,Y 166.114,Z 496.226,A -85,B 0,C 180,E1 -23966.883,E2 -23966.883} C_VEL
LIN {X 0,Y 167.437,Z 497.999,A -85,B 0,C 180,E1 -23967.928,E2 -23967.928} C_VEL
LIN {X 0,Y 170.332,Z 502.666,A -85,B 0,C 180,E1 -23970.19,E2 -23970.19} C_VEL
LIN {X 0,Y 173.96,Z 509.46,A -85,B 0,C 180,E1 -23972.963,E2 -23972.963} C_VEL
LIN {X 0,Y 177.649,Z 517.204,A -85,B 0,C 180,E1 -23975.787,E2 -23975.787} C_VEL
LIN {X 0,Y 180.507,Z 524.642,A -85,B 0,C 180,E1 -23978.177,E2 -23978.177} C_VEL
LIN {X 0,Y 181.734,Z 535.883,A -85,B 0,C 180,E1 -23980.737,E2 -23980.737} C_VEL
LIN {X 0,Y 182.053,Z 547.512,A -85,B 0,C 180,E1 -23983.426,E2 -23983.426} C_VEL
LIN {X 0,Y 181.292,Z 558.773,A -85,B 0,C 180,E1 -23986.125,E2 -23986.125} C_VEL
LIN {X 0,Y 180.488,Z 565.006,A -85,B 0,C 180,E1 -23987.718,E2 -23987.718} C_VEL
LIN {X 0,Y 176.173,Z 575.334,A -85,B 0,C 180,E1 -23989.964,E2 -23989.964} C_VEL
LIN {X 0,Y 171.076,Z 585.599,A -85,B 0,C 180,E1 -23992.703,E2 -23992.703} C_VEL
LIN {X 0,Y 166.199,Z 594.862,A -85,B 0,C 180,E1 -23995.924,E2 -23995.924} C_VEL
LIN {X 0,Y 161.042,Z 603.667,A -85,B 0,C 180,E1 -23999.876,E2 -23999.876} C_VEL
LIN {X 0,Y 157.249,Z 609.879,A -85,B 0,C 180,E1 -24003.453,E2 -24003.453} C_VEL
LIN {X 0,Y 154.357,Z 614.966,A -85,B 0,C 180,E1 -24007.231,E2 -24007.231} C_VEL
LIN {X 0,Y 151.024,Z 620.299,A -85,B 0,C 180,E1 -24012.393,E2 -24012.393} C_VEL
LIN {X 0,Y 149.389,Z 623.242,A -85,B 0,C 180,E1 -24016.395,E2 -24016.395} C_VEL
LIN {X 0,Y 148.028,Z 625.956,A -85,B 0,C 180,E1 -24021.811,E2 -24021.811} C_VEL
LIN {X 0,Y 147.571,Z 627.312,A -85,B 0,C 180,E1 -24027.27,E2 -24027.27} C_VEL
LIN {X 0,Y 147.597,Z 627.466,A -85,B 0,C 180,E1 -24030.613,E2 -24030.613} C_VEL
LIN {X 0,Y 147.703,Z 626.847,A -85,B 0,C 180,E1 -24035.461,E2 -24035.461} C_VEL
LIN {X 0,Y 148.591,Z 624.856,A -85,B 0,C 180,E1 -24040.906,E2 -24040.906} C_VEL
LIN {X 0,Y 150.351,Z 621.478,A -85,B 0,C 180,E1 -24046.288,E2 -24046.288} C_VEL
LIN {X 0,Y 153.369,Z 616.608,A -85,B 0,C 180,E1 -24051.506,E2 -24051.506} C_VEL
LIN {X 0,Y 156.282,Z 611.883,A -85,B 0,C 180,E1 -24055.291,E2 -24055.291} C_VEL
LIN {X 0,Y 159.718,Z 606.138,A -85,B 0,C 180,E1 -24058.949,E2 -24058.949} C_VEL
LIN {X 0,Y 164.578,Z 597.869,A -85,B 0,C 180,E1 -24062.988,E2 -24062.988} C_VEL
LIN {X 0,Y 169.295,Z 589.237,A -85,B 0,C 180,E1 -24066.268,E2 -24066.268} C_VEL
LIN {X 0,Y 174.614,Z 578.771,A -85,B 0,C 180,E1 -24069.34,E2 -24069.34} C_VEL
LIN {X 0,Y 179.357,Z 568.202,A -85,B 0,C 180,E1 -24071.77,E2 -24071.77} C_VEL
LIN {X 0,Y 180.585,Z 565.119,A -85,B 0,C 180,E1 -24072.4,E2 -24072.4} C_VEL
LIN {X 0,Y 181.915,Z 553.002,A -85,B 0,C 180,E1 -24075.429,E2 -24075.429} C_VEL
LIN {X 0,Y 182.105,Z 542.135,A -85,B 0,C 180,E1 -24077.998,E2 -24077.998} C_VEL
LIN {X 0,Y 181.478,Z 531.451,A -85,B 0,C 180,E1 -24080.427,E2 -24080.427} C_VEL
LIN {X 0,Y 180.408,Z 524.165,A -85,B 0,C 180,E1 -24082.152,E2 -24082.152} C_VEL
LIN {X 0,Y 176.905,Z 515.576,A -85,B 0,C 180,E1 -24085,E2 -24085} C_VEL
LIN {X 0,Y 174.002,Z 509.427,A -85,B 0,C 180,E1 -24087.255,E2 -24087.255} C_VEL
LIN {X 0,Y 173.232,Z 510.101,A -85,B 0,C 180,E1 -24087.568,E2 -24087.568} C_VEL
LIN {X 0,Y 168.892,Z 514.526,A -85,B 0,C 180,E1 -24089.266,E2 -24089.266} C_VEL
LIN {X 0,Y 165.938,Z 516.488,A -85,B 0,C 180,E1 -24090.678,E2 -24090.678} C_VEL
LIN {X 0,Y 164.379,Z 516.821,A -85,B 0,C 180,E1 -24091.598,E2 -24091.598} C_VEL
LIN {X 0,Y 160.461,Z 521.474,A -85,B 0,C 180,E1 -24093.236,E2 -24093.236} C_VEL
LIN {X 0,Y 156.928,Z 524.632,A -85,B 0,C 180,E1 -24095.087,E2 -24095.087} C_VEL
LIN {X 0,Y 155.541,Z 525.311,A -85,B 0,C 180,E1 -24096.005,E2 -24096.005} C_VEL
LIN {X 0,Y 154.315,Z 524.651,A -85,B 0,C 180,E1 -24097.313,E2 -24097.313} C_VEL
LIN {X 0,Y 152.707,Z 532.559,A -85,B 0,C 180,E1 -24100.508,E2 -24100.508} C_VEL
LIN {X 0,Y 150.828,Z 542.334,A -85,B 0,C 180,E1 -24105.15,E2 -24105.15} C_VEL
LIN {X 0,Y 149.66,Z 550.83,A -85,B 0,C 180,E1 -24110.012,E2 -24110.012} C_VEL
LIN {X 0,Y 149.156,Z 557.603,A -85,B 0,C 180,E1 -24114.592,E2 -24114.592} C_VEL
LIN {X 0,Y 148.872,Z 564.15,A -85,B 0,C 180,E1 -24120,E2 -24120} C_VEL
LIN {X 0,Y 150.104,Z 570.669,A -85,B 0,C 180,E1 -24126.722,E2 -24126.722} C_VEL
LIN {X 0,Y 153.079,Z 575.45,A -85,B 0,C 180,E1 -24133.271,E2 -24133.271} C_VEL
LIN {X 0,Y 156.528,Z 578.22,A -85,B 0,C 180,E1 -24138.318,E2 -24138.318} C_VEL
LIN {X 0,Y 160.996,Z 580.036,A -85,B 0,C 180,E1 -24143.134,E2 -24143.134} C_VEL
LIN {X 0,Y 166.67,Z 580.971,A -85,B 0,C 180,E1 -24147.635,E2 -24147.635} C_VEL
LIN {X 0,Y 173.469,Z 581.091,A -85,B 0,C 180,E1 -24151.782,E2 -24151.782} C_VEL
LIN {X 0,Y 181.279,Z 580.31,A -85,B 0,C 180,E1 -24155.558,E2 -24155.558} C_VEL
LIN {X 0,Y 194.684,Z 577.661,A -85,B 0,C 180,E1 -24160.526,E2 -24160.526} C_VEL
LIN {X 0,Y 198.726,Z 576.694,A -85,B 0,C 180,E1 -24162.04,E2 -24162.04} C_VEL
LIN {X 0,Y 187.024,Z 582.654,A -85,B 0,C 180,E1 -24165.957,E2 -24165.957} C_VEL
LIN {X 0,Y 175.783,Z 587.826,A -85,B 0,C 180,E1 -24170.231,E2 -24170.231} C_VEL
LIN {X 0,Y 169.084,Z 590.748,A -85,B 0,C 180,E1 -24173.494,E2 -24173.494} C_VEL
LIN {X 0,Y 164.117,Z 599.892,A -85,B 0,C 180,E1 -24176.907,E2 -24176.907} C_VEL
LIN {X 0,Y 159.26,Z 608.257,A -85,B 0,C 180,E1 -24180.96,E2 -24180.96} C_VEL
LIN {X 0,Y 155.879,Z 614.04,A -85,B 0,C 180,E1 -24184.61,E2 -24184.61} C_VEL
LIN {X 0,Y 152.991,Z 618.863,A -85,B 0,C 180,E1 -24188.438,E2 -24188.438} C_VEL
LIN {X 0,Y 150.051,Z 623.795,A -85,B 0,C 180,E1 -24193.679,E2 -24193.679} C_VEL
LIN {X 0,Y 148.383,Z 627.225,A -85,B 0,C 180,E1 -24199.079,E2 -24199.079} C_VEL
LIN {X 0,Y 147.686,Z 629.255,A -85,B 0,C 180,E1 -24204.539,E2 -24204.539} C_VEL
LIN {X 0,Y 147.656,Z 629.925,A -85,B 0,C 180,E1 -24210,E2 -24210} C_VEL
LIN {X 0,Y 147.685,Z 629.236,A -85,B 0,C 180,E1 -24215.461,E2 -24215.461} C_VEL
LIN {X 0,Y 148.375,Z 627.191,A -85,B 0,C 180,E1 -24220.922,E2 -24220.922} C_VEL
LIN {X 0,Y 150.039,Z 623.74,A -85,B 0,C 180,E1 -24226.323,E2 -24226.323} C_VEL
LIN {X 0,Y 150.57,Z 622.844,A -85,B 0,C 180,E1 -24227.441,E2 -24227.441} C_VEL
LIN {X 0,Y 151.036,Z 621.053,A -85,B 0,C 180,E1 -24229.574,E2 -24229.574} C_VEL
LIN {X 0,Y 150.335,Z 617.712,A -85,B 0,C 180,E1 -24233.12,E2 -24233.12} C_VEL
LIN {X 0,Y 150.051,Z 613.759,A -85,B 0,C 180,E1 -24236.602,E2 -24236.602} C_VEL
LIN {X 0,Y 151.14,Z 611.007,A -85,B 0,C 180,E1 -24238.555,E2 -24238.555} C_VEL
LIN {X 0,Y 155.847,Z 603.494,A -85,B 0,C 180,E1 -24242.762,E2 -24242.762} C_VEL
LIN {X 0,Y 160.539,Z 595.507,A -85,B 0,C 180,E1 -24246.228,E2 -24246.228} C_VEL
LIN {X 0,Y 165.939,Z 585.864,A -85,B 0,C 180,E1 -24249.442,E2 -24249.442} C_VEL
LIN {X 0,Y 171.048,Z 575.357,A -85,B 0,C 180,E1 -24252.206,E2 -24252.206} C_VEL
LIN {X 0,Y 172.399,Z 571.219,A -85,B 0,C 180,E1 -24253.276,E2 -24253.276} C_VEL
LIN {X 0,Y 175.087,Z 559.095,A -85,B 0,C 180,E1 -24256.263,E2 -24256.263} C_VEL
LIN {X 0,Y 176.321,Z 551.334,A -85,B 0,C 180,E1 -24257.985,E2 -24257.985} C_VEL
LIN {X 0,Y 176.452,Z 541.073,A -85,B 0,C 180,E1 -24260.411,E2 -24260.411} C_VEL
LIN {X 0,Y 175.525,Z 530.039,A -85,B 0,C 180,E1 -24263.088,E2 -24263.088} C_VEL
LIN {X 0,Y 173.662,Z 519.266,A -85,B 0,C 180,E1 -24265.84,E2 -24265.84} C_VEL
LIN {X 0,Y 171.729,Z 512.213,A -85,B 0,C 180,E1 -24267.858,E2 -24267.858} C_VEL
LIN {X 0,Y 168.468,Z 505.475,A -85,B 0,C 180,E1 -24270.562,E2 -24270.562} C_VEL
LIN {X 0,Y 166.275,Z 501.535,A -85,B 0,C 180,E1 -24272.379,E2 -24272.379} C_VEL
LIN {X 0,Y 163.312,Z 496.291,A -85,B 0,C 180,E1 -24275.022,E2 -24275.022} C_VEL
LIN {X 0,Y 158.83,Z 490.831,A -85,B 0,C 180,E1 -24279.574,E2 -24279.574} C_VEL
LIN {X 0,Y 157.715,Z 488.115,A -85,B 0,C 180,E1 -24284.492,E2 -24284.492} C_VEL
LIN {X 0,Y 156.906,Z 486.137,A -85,B 0,C 180,E1 -24289.679,E2 -24289.679} C_VEL
LIN {X 0,Y 156.32,Z 485.132,A -85,B 0,C 180,E1 -24294.841,E2 -24294.841} C_VEL
LIN {X 0,Y 156.309,Z 484.778,A -85,B 0,C 180,E1 -24300,E2 -24300} C_VEL
LIN {X 0,Y 155.91,Z 485.817,A -85,B 0,C 180,E1 -24305.173,E2 -24305.173} C_VEL
LIN {X 0,Y 156.007,Z 487.458,A -85,B 0,C 180,E1 -24310.381,E2 -24310.381} C_VEL
LIN {X 0,Y 156.136,Z 489.92,A -85,B 0,C 180,E1 -24315.669,E2 -24315.669} C_VEL
LIN {X 0,Y 156.416,Z 491.443,A -85,B 0,C 180,E1 -24318.037,E2 -24318.037} C_VEL
LIN {X 0,Y 159.723,Z 496.38,A -85,B 0,C 180,E1 -24321.963,E2 -24321.963} C_VEL
LIN {X 0,Y 161.203,Z 498.11,A -85,B 0,C 180,E1 -24323.429,E2 -24323.429} C_VEL
LIN {X 0,Y 164.25,Z 502.956,A -85,B 0,C 180,E1 -24326.355,E2 -24326.355} C_VEL
LIN {X 0,Y 168.036,Z 509.763,A -85,B 0,C 180,E1 -24329.745,E2 -24329.745} C_VEL
LIN {X 0,Y 170.691,Z 515.291,A -85,B 0,C 180,E1 -24332.1,E2 -24332.1} C_VEL
LIN {X 0,Y 173.817,Z 522.633,A -85,B 0,C 180,E1 -24334.917,E2 -24334.917} C_VEL
LIN {X 0,Y 175.831,Z 528.509,A -85,B 0,C 180,E1 -24336.927,E2 -24336.927} C_VEL
LIN {X 0,Y 176.702,Z 539.116,A -85,B 0,C 180,E1 -24339.522,E2 -24339.522} C_VEL
LIN {X 0,Y 176.625,Z 550.692,A -85,B 0,C 180,E1 -24342.357,E2 -24342.357} C_VEL
LIN {X 0,Y 175.341,Z 562.814,A -85,B 0,C 180,E1 -24345.459,E2 -24345.459} C_VEL
LIN {X 0,Y 174.846,Z 566.092,A -85,B 0,C 180,E1 -24346.346,E2 -24346.346} C_VEL
LIN {X 0,Y 170.307,Z 576.43,A -85,B 0,C 180,E1 -24348.68,E2 -24348.68} C_VEL
LIN {X 0,Y 164.576,Z 587.301,A -85,B 0,C 180,E1 -24351.742,E2 -24351.742} C_VEL
LIN {X 0,Y 159.537,Z 596.265,A -85,B 0,C 180,E1 -24355.063,E2 -24355.063} C_VEL
LIN {X 0,Y 154.199,Z 604.828,A -85,B 0,C 180,E1 -24359.153,E2 -24359.153} C_VEL
LIN {X 0,Y 149.811,Z 611.725,A -85,B 0,C 180,E1 -24363.534,E2 -24363.534} C_VEL
LIN {X 0,Y 146.823,Z 616.493,A -85,B 0,C 180,E1 -24367.484,E2 -24367.484} C_VEL
LIN {X 0,Y 143.563,Z 621.411,A -85,B 0,C 180,E1 -24372.919,E2 -24372.919} C_VEL
LIN {X 0,Y 141.617,Z 624.831,A -85,B 0,C 180,E1 -24378.55,E2 -24378.55} C_VEL
LIN {X 0,Y 140.635,Z 626.859,A -85,B 0,C 180,E1 -24384.264,E2 -24384.264} C_VEL
LIN {X 0,Y 140.524,Z 627.548,A -85,B 0,C 180,E1 -24390,E2 -24390} C_VEL
LIN {X 0,Y 140.635,Z 626.905,A -85,B 0,C 180,E1 -24395.736,E2 -24395.736} C_VEL
LIN {X 0,Y 141.613,Z 624.914,A -85,B 0,C 180,E1 -24401.45,E2 -24401.45} C_VEL
LIN {X 0,Y 143.503,Z 621.536,A -85,B 0,C 180,E1 -24407.088,E2 -24407.088} C_VEL
LIN {X 0,Y 146.772,Z 616.664,A -85,B 0,C 180,E1 -24412.524,E2 -24412.524} C_VEL
LIN {X 0,Y 149.85,Z 611.939,A -85,B 0,C 180,E1 -24416.459,E2 -24416.459} C_VEL
LIN {X 0,Y 154.198,Z 605.09,A -85,B 0,C 180,E1 -24420.847,E2 -24420.847} C_VEL
LIN {X 0,Y 159.437,Z 596.584,A -85,B 0,C 180,E1 -24424.963,E2 -24424.963} C_VEL
LIN {X 0,Y 164.514,Z 587.681,A -85,B 0,C 180,E1 -24428.275,E2 -24428.275} C_VEL
LIN {X 0,Y 170.162,Z 576.895,A -85,B 0,C 180,E1 -24431.363,E2 -24431.363} C_VEL
LIN {X 0,Y 174.555,Z 567.195,A -85,B 0,C 180,E1 -24433.554,E2 -24433.554} C_VEL
LIN {X 0,Y 175.355,Z 563.407,A -85,B 0,C 180,E1 -24434.536,E2 -24434.536} C_VEL
LIN {X 0,Y 176.609,Z 552.213,A -85,B 0,C 180,E1 -24437.429,E2 -24437.429} C_VEL
LIN {X 0,Y 176.9,Z 541.287,A -85,B 0,C 180,E1 -24440.106,E2 -24440.106} C_VEL
LIN {X 0,Y 176.132,Z 529.656,A -85,B 0,C 180,E1 -24442.943,E2 -24442.943} C_VEL
LIN {X 0,Y 175.408,Z 526.964,A -85,B 0,C 180,E1 -24443.773,E2 -24443.773} C_VEL
LIN {X 0,Y 172.164,Z 518.216,A -85,B 0,C 180,E1 -24446.908,E2 -24446.908} C_VEL
LIN {X 0,Y 167.239,Z 522.003,A -85,B 0,C 180,E1 -24448.841,E2 -24448.841} C_VEL
LIN {X 0,Y 164.057,Z 523.578,A -85,B 0,C 180,E1 -24450.397,E2 -24450.397} C_VEL
LIN {X 0,Y 159.122,Z 528.517,A -85,B 0,C 180,E1 -24452.371,E2 -24452.371} C_VEL
LIN {X 0,Y 157.019,Z 530.151,A -85,B 0,C 180,E1 -24453.411,E2 -24453.411} C_VEL
LIN {X 0,Y 151.683,Z 532.765,A -85,B 0,C 180,E1 -24456.806,E2 -24456.806} C_VEL
LIN {X 0,Y 147.803,Z 536.147,A -85,B 0,C 180,E1 -24459.107,E2 -24459.107} C_VEL
LIN {X 0,Y 146.217,Z 537.136,A -85,B 0,C 180,E1 -24460.339,E2 -24460.339} C_VEL
LIN {X 0,Y 145.02,Z 537.282,A -85,B 0,C 180,E1 -24461.639,E2 -24461.639} C_VEL
LIN {X 0,Y 144.717,Z 536.74,A -85,B 0,C 180,E1 -24462.33,E2 -24462.33} C_VEL
LIN {X 0,Y 143.133,Z 545.962,A -85,B 0,C 180,E1 -24467.235,E2 -24467.235} C_VEL
LIN {X 0,Y 142.219,Z 553.44,A -85,B 0,C 180,E1 -24471.965,E2 -24471.965} C_VEL
LIN {X 0,Y 141.97,Z 558.59,A -85,B 0,C 180,E1 -24475.741,E2 -24475.741} C_VEL
LIN {X 0,Y 141.887,Z 565.124,A -85,B 0,C 180,E1 -24481.419,E2 -24481.419} C_VEL
LIN {X 0,Y 143.574,Z 571.612,A -85,B 0,C 180,E1 -24488.444,E2 -24488.444} C_VEL
LIN {X 0,Y 146.191,Z 575.611,A -85,B 0,C 180,E1 -24493.908,E2 -24493.908} C_VEL
LIN {X 0,Y 149.83,Z 578.612,A -85,B 0,C 180,E1 -24499.168,E2 -24499.168} C_VEL
LIN {X 0,Y 154.538,Z 580.754,A -85,B 0,C 180,E1 -24504.16,E2 -24504.16} C_VEL
LIN {X 0,Y 160.495,Z 582.021,A -85,B 0,C 180,E1 -24508.795,E2 -24508.795} C_VEL
LIN {X 0,Y 167.599,Z 582.407,A -85,B 0,C 180,E1 -24513.034,E2 -24513.034} C_VEL
LIN {X 0,Y 175.735,Z 582.03,A -85,B 0,C 180,E1 -24516.861,E2 -24516.861} C_VEL
LIN {X 0,Y 184.793,Z 580.803,A -85,B 0,C 180,E1 -24520.281,E2 -24520.281} C_VEL
LIN {X 0,Y 189.595,Z 579.893,A -85,B 0,C 180,E1 -24521.854,E2 -24521.854} C_VEL
LIN {X 0,Y 184.497,Z 582.265,A -85,B 0,C 180,E1 -24523.634,E2 -24523.634} C_VEL
LIN {X 0,Y 170.385,Z 588.012,A -85,B 0,C 180,E1 -24528.703,E2 -24528.703} C_VEL
LIN {X 0,Y 163.427,Z 590.698,A -85,B 0,C 180,E1 -24532.012,E2 -24532.012} C_VEL
LIN {X 0,Y 158.191,Z 599.84,A -85,B 0,C 180,E1 -24535.497,E2 -24535.497} C_VEL
LIN {X 0,Y 153.052,Z 608.203,A -85,B 0,C 180,E1 -24539.661,E2 -24539.661} C_VEL
LIN {X 0,Y 149.191,Z 614.41,A -85,B 0,C 180,E1 -24543.741,E2 -24543.741} C_VEL
LIN {X 0,Y 145.497,Z 620.221,A -85,B 0,C 180,E1 -24548.76,E2 -24548.76} C_VEL
LIN {X 0,Y 143.209,Z 623.737,A -85,B 0,C 180,E1 -24552.875,E2 -24552.875} C_VEL
LIN {X 0,Y 141.389,Z 627.167,A -85,B 0,C 180,E1 -24558.532,E2 -24558.532} C_VEL
LIN {X 0,Y 140.616,Z 629.197,A -85,B 0,C 180,E1 -24564.263,E2 -24564.263} C_VEL
LIN {X 0,Y 140.56,Z 629.867,A -85,B 0,C 180,E1 -24570,E2 -24570} C_VEL
LIN {X 0,Y 140.615,Z 629.177,A -85,B 0,C 180,E1 -24575.737,E2 -24575.737} C_VEL
LIN {X 0,Y 141.382,Z 627.132,A -85,B 0,C 180,E1 -24581.469,E2 -24581.469} C_VEL
LIN {X 0,Y 143.196,Z 623.681,A -85,B 0,C 180,E1 -24587.126,E2 -24587.126} C_VEL
LIN {X 0,Y 146.303,Z 618.725,A -85,B 0,C 180,E1 -24592.6,E2 -24592.6} C_VEL
LIN {X 0,Y 149.197,Z 614.028,A -85,B 0,C 180,E1 -24596.491,E2 -24596.491} C_VEL
LIN {X 0,Y 151.14,Z 611.007,A -85,B 0,C 180,E1 -24598.555,E2 -24598.555} C_VEL
LIN {X 0,Y 152.375,Z 608.14,A -85,B 0,C 180,E1 -24600.442,E2 -24600.442} C_VEL
LIN {X 0,Y 153.033,Z 603.136,A -85,B 0,C 180,E1 -24603.655,E2 -24603.655} C_VEL
LIN {X 0,Y 154.014,Z 597.724,A -85,B 0,C 180,E1 -24606.726,E2 -24606.726} C_VEL
LIN {X 0,Y 155.689,Z 594.039,A -85,B 0,C 180,E1 -24608.331,E2 -24608.331} C_VEL
LIN {X 0,Y 161.5,Z 584.04,A -85,B 0,C 180,E1 -24611.578,E2 -24611.578} C_VEL
LIN {X 0,Y 166.026,Z 574.854,A -85,B 0,C 180,E1 -24613.977,E2 -24613.977} C_VEL
LIN {X 0,Y 169.121,Z 563.196,A -85,B 0,C 180,E1 -24617.09,E2 -24617.09} C_VEL
LIN {X 0,Y 170.968,Z 553.796,A -85,B 0,C 180,E1 -24619.289,E2 -24619.289} C_VEL
LIN {X 0,Y 171.45,Z 544.541,A -85,B 0,C 180,E1 -24621.623,E2 -24621.623} C_VEL
LIN {X 0,Y 170.947,Z 533.609,A -85,B 0,C 180,E1 -24624.423,E2 -24624.423} C_VEL
LIN {X 0,Y 169.283,Z 521.892,A -85,B 0,C 180,E1 -24627.601,E2 -24627.601} C_VEL
LIN {X 0,Y 168.006,Z 516.94,A -85,B 0,C 180,E1 -24629.174,E2 -24629.174} C_VEL
LIN {X 0,Y 164.968,Z 510.009,A -85,B 0,C 180,E1 -24632.141,E2 -24632.141} C_VEL
LIN {X 0,Y 163.193,Z 506.554,A -85,B 0,C 180,E1 -24633.891,E2 -24633.891} C_VEL
LIN {X 0,Y 161.083,Z 502.461,A -85,B 0,C 180,E1 -24636.028,E2 -24636.028} C_VEL
LIN {X 0,Y 156.726,Z 497.092,A -85,B 0,C 180,E1 -24640.739,E2 -24640.739} C_VEL
LIN {X 0,Y 151.591,Z 490.976,A -85,B 0,C 180,E1 -24648.975,E2 -24648.975} C_VEL
LIN {X 0,Y 151.207,Z 490.199,A -85,B 0,C 180,E1 -24651.985,E2 -24651.985} C_VEL
LIN {X 0,Y 150.808,Z 489.437,A -85,B 0,C 180,E1 -24657.329,E2 -24657.329} C_VEL
LIN {X 0,Y 150.842,Z 489.332,A -85,B 0,C 180,E1 -24660,E2 -24660} C_VEL
LIN {X 0,Y 150.374,Z 490.332,A -85,B 0,C 180,E1 -24665.364,E2 -24665.364} C_VEL
LIN {X 0,Y 150.455,Z 491.417,A -85,B 0,C 180,E1 -24668.732,E2 -24668.732} C_VEL
LIN {X 0,Y 154.906,Z 498.185,A -85,B 0,C 180,E1 -24677.311,E2 -24677.311} C_VEL
LIN {X 0,Y 158.144,Z 503.211,A -85,B 0,C 180,E1 -24681.508,E2 -24681.508} C_VEL
LIN {X 0,Y 159.177,Z 504.637,A -85,B 0,C 180,E1 -24682.641,E2 -24682.641} C_VEL
LIN {X 0,Y 162.329,Z 510.269,A -85,B 0,C 180,E1 -24686.086,E2 -24686.086} C_VEL
LIN {X 0,Y 164.949,Z 515.601,A -85,B 0,C 180,E1 -24688.816,E2 -24688.816} C_VEL
LIN {X 0,Y 167.073,Z 520.48,A -85,B 0,C 180,E1 -24691.018,E2 -24691.018} C_VEL
LIN {X 0,Y 169.396,Z 526.63,A -85,B 0,C 180,E1 -24693.515,E2 -24693.515} C_VEL
LIN {X 0,Y 171.169,Z 532.261,A -85,B 0,C 180,E1 -24695.595,E2 -24695.595} C_VEL
LIN {X 0,Y 171.666,Z 539.199,A -85,B 0,C 180,E1 -24697.447,E2 -24697.447} C_VEL
LIN {X 0,Y 171.386,Z 551.891,A -85,B 0,C 180,E1 -24700.735,E2 -24700.735} C_VEL
LIN {X 0,Y 169.8,Z 564.132,A -85,B 0,C 180,E1 -24704.017,E2 -24704.017} C_VEL
LIN {X 0,Y 169.091,Z 567.752,A -85,B 0,C 180,E1 -24705.043,E2 -24705.043} C_VEL
LIN {X 0,Y 164.007,Z 578.416,A -85,B 0,C 180,E1 -24707.552,E2 -24707.552} C_VEL
LIN {X 0,Y 158.124,Z 588.962,A -85,B 0,C 180,E1 -24710.702,E2 -24710.702} C_VEL
LIN {X 0,Y 152.899,Z 597.66,A -85,B 0,C 180,E1 -24714.122,E2 -24714.122} C_VEL
LIN {X 0,Y 147.377,Z 605.989,A -85,B 0,C 180,E1 -24718.361,E2 -24718.361} C_VEL
LIN {X 0,Y 143.062,Z 612.395,A -85,B 0,C 180,E1 -24722.723,E2 -24722.723} C_VEL
LIN {X 0,Y 139.277,Z 617.96,A -85,B 0,C 180,E1 -24727.762,E2 -24727.762} C_VEL
LIN {X 0,Y 136.752,Z 621.471,A -85,B 0,C 180,E1 -24732.04,E2 -24732.04} C_VEL
LIN {X 0,Y 134.633,Z 624.891,A -85,B 0,C 180,E1 -24737.948,E2 -24737.948} C_VEL
LIN {X 0,Y 133.564,Z 626.918,A -85,B 0,C 180,E1 -24743.959,E2 -24743.959} C_VEL
LIN {X 0,Y 133.449,Z 627.607,A -85,B 0,C 180,E1 -24750,E2 -24750} C_VEL
LIN {X 0,Y 133.564,Z 626.963,A -85,B 0,C 180,E1 -24756.041,E2 -24756.041} C_VEL
LIN {X 0,Y 134.626,Z 624.972,A -85,B 0,C 180,E1 -24762.053,E2 -24762.053} C_VEL
LIN {X 0,Y 136.69,Z 621.593,A -85,B 0,C 180,E1 -24767.968,E2 -24767.968} C_VEL
LIN {X 0,Y 140.224,Z 616.721,A -85,B 0,C 180,E1 -24773.638,E2 -24773.638} C_VEL
LIN {X 0,Y 144.678,Z 610.206,A -85,B 0,C 180,E1 -24779.063,E2 -24779.063} C_VEL
LIN {X 0,Y 149.625,Z 602.931,A -85,B 0,C 180,E1 -24783.498,E2 -24783.498} C_VEL
LIN {X 0,Y 155.363,Z 593.858,A -85,B 0,C 180,E1 -24787.639,E2 -24787.639} C_VEL
LIN {X 0,Y 160.905,Z 584.36,A -85,B 0,C 180,E1 -24790.932,E2 -24790.932} C_VEL
LIN {X 0,Y 166.724,Z 573.351,A -85,B 0,C 180,E1 -24793.839,E2 -24793.839} C_VEL
LIN {X 0,Y 169.341,Z 567.252,A -85,B 0,C 180,E1 -24795.251,E2 -24795.251} C_VEL
LIN {X 0,Y 171.064,Z 556.378,A -85,B 0,C 180,E1 -24798.25,E2 -24798.25} C_VEL
LIN {X 0,Y 171.769,Z 545.81,A -85,B 0,C 180,E1 -24801.023,E2 -24801.023} C_VEL
